# B&R Automation Studio project Assembly_and_ST (part 2)

#### providePellet.st
```iecst
ACTION providePellet:
		(*************************************************************************************************)
		(*************************************************************************************************)
		(* State Machine *)
	CASE gAssemblyModule.skill.providePellet.state.stateMachine.operationalState OF
		(*************************************************************************************************)
		(* RESETTING *)
		RESETTING:
			(*gAssemblyModule.skill.providePellet.state.stateMachine.stateTransition.reset := FALSE;*)

			IF gAssemblyModule.skill.providePellet.state.stateMachine.stateTransition.abort THEN
				gAssemblyModule.skill.providePellet.state.stateMachine.operationalState := ABORTING;

			ELSIF gAssemblyModule.skill.providePellet.state.stateMachine.stateTransition.stop THEN
				gAssemblyModule.skill.providePellet.state.stateMachine.operationalState := STOPPING;

			ELSE
				providePellet_Resetting;

			END_IF;

			(*************************************************************************************************)
			(* IDLE *)
		IDLE:

			gAssemblyModule.skill.providePellet.state.stateMachine.stateTransition.reset := FALSE;

			IF gAssemblyModule.skill.providePellet.state.stateMachine.stateTransition.abort THEN
				gAssemblyModule.skill.providePellet.state.stateMachine.operationalState := ABORTING;

			ELSIF gAssemblyModule.skill.providePellet.state.stateMachine.stateTransition.stop THEN
				gAssemblyModule.skill.providePellet.state.stateMachine.operationalState := STOPPING;

			ELSE
				providePellet_Idle;

			END_IF;

			(*************************************************************************************************)
			(* STARTING *)
		STARTING:
			(*gAssemblyModule.skill.providePellet.state.stateMachine.stateTransition.start := FALSE;*)

			IF gAssemblyModule.skill.providePellet.state.stateMachine.stateTransition.abort THEN
				gAssemblyModule.skill.providePellet.state.stateMachine.operationalState := ABORTING;

			ELSIF gAssemblyModule.skill.providePellet.state.stateMachine.stateTransition.stop THEN
				gAssemblyModule.skill.providePellet.state.stateMachine.operationalState := STOPPING;

			ELSE
				providePellet_Starting;

			END_IF;

			(*************************************************************************************************)
			(* RUNNING *)
		RUNNING:

			gAssemblyModule.skill.providePellet.state.stateMachine.stateTransition.start := FALSE;

			IF gAssemblyModule.skill.providePellet.state.stateMachine.stateTransition.abort THEN
				gAssemblyModule.skill.providePellet.state.stateMachine.operationalState := ABORTING;

			ELSIF gAssemblyModule.skill.providePellet.state.stateMachine.stateTransition.stop THEN
				gAssemblyModule.skill.providePellet.state.stateMachine.operationalState := STOPPING;

			ELSIF gAssemblyModule.skill.providePellet.state.stateMachine.stateTransition.hold THEN
				gAssemblyModule.skill.providePellet.state.stateMachine.operationalState := HOLDING;

			ELSIF gAssemblyModule.skill.providePellet.state.stateMachine.stateTransition.suspend THEN
				gAssemblyModule.skill.providePellet.state.stateMachine.operationalState := SUSPENDING;

			ELSIF gAssemblyModule.skill.providePellet.state.stateMachine.stateTransition.pause THEN
				gAssemblyModule.skill.providePellet.state.stateMachine.operationalState := PAUSING;

			ELSE
				providePellet_Running;

			END_IF;

			(*************************************************************************************************)
			(* PAUSING *)
		PAUSING:
			(*	gAssemblyModule.skill.providePellet.state.stateMachine.stateTransition.pause := FALSE;*)

			IF gAssemblyModule.skill.providePellet.state.stateMachine.stateTransition.abort THEN
				gAssemblyModule.skill.providePellet.state.stateMachine.operationalState := ABORTING;

			ELSIF gAssemblyModule.skill.providePellet.state.stateMachine.stateTransition.stop THEN
				gAssemblyModule.skill.providePellet.state.stateMachine.operationalState := STOPPING;

			ELSIF gAssemblyModule.skill.providePellet.state.stateMachine.stateTransition.hold THEN
				//gAssemblyModule.skill.providePellet.state.stateMachine.operationalState := HOLDING;

			ELSIF gAssemblyModule.skill.providePellet.state.stateMachine.stateTransition.suspend THEN
				//gAssemblyModule.skill.providePellet.state.stateMachine.operationalState := SUSPENDING;

			ELSE
				providePellet_Pausing;
			END_IF;

			(*************************************************************************************************)
			(* PAUSED *)
		PAUSED:

			gAssemblyModule.skill.providePellet.state.stateMachine.stateTransition.pause := FALSE;

			IF gAssemblyModule.skill.providePellet.state.stateMachine.stateTransition.abort THEN
				gAssemblyModule.skill.providePellet.state.stateMachine.operationalState := ABORTING;

			ELSIF gAssemblyModule.skill.providePellet.state.stateMachine.stateTransition.stop THEN
				gAssemblyModule.skill.providePellet.state.stateMachine.operationalState := STOPPING;

			ELSIF gAssemblyModule.skill.providePellet.state.stateMachine.stateTransition.hold THEN
				//gAssemblyModule.skill.providePellet.state.stateMachine.operationalState := HOLDING;

			ELSIF gAssemblyModule.skill.providePellet.state.stateMachine.stateTransition.suspend THEN
				//gAssemblyModule.skill.providePellet.state.stateMachine.operationalState := SUSPENDING;

			ELSE
				providePellet_Paused;

			END_IF;

			(*************************************************************************************************)
			(* SUSPENDING *)
		SUSPENDING:
			(*gAssemblyModule.skill.providePellet.state.stateMachine.stateTransition.suspend := FALSE;*)

			IF gAssemblyModule.skill.providePellet.state.stateMachine.stateTransition.abort THEN
				gAssemblyModule.skill.providePellet.state.stateMachine.operationalState := ABORTING;

			ELSIF gAssemblyModule.skill.providePellet.state.stateMachine.stateTransition.stop THEN
				gAssemblyModule.skill.providePellet.state.stateMachine.operationalState := STOPPING;

			ELSIF gAssemblyModule.skill.providePellet.state.stateMachine.stateTransition.hold THEN
				//gAssemblyModule.skill.providePellet.state.stateMachine.operationalState := HOLDING;

			ELSE
				providePellet_Suspending;

			END_IF;

			(*************************************************************************************************)
			(* SUSPENDED *)
		SUSPENDED:

			gAssemblyModule.skill.providePellet.state.stateMachine.stateTransition.suspend := FALSE;

			IF gAssemblyModule.skill.providePellet.state.stateMachine.stateTransition.abort THEN
				gAssemblyModule.skill.providePellet.state.stateMachine.operationalState := ABORTING;

			ELSIF gAssemblyModule.skill.providePellet.state.stateMachine.stateTransition.stop THEN
				gAssemblyModule.skill.providePellet.state.stateMachine.operationalState := STOPPING;

			ELSIF gAssemblyModule.skill.providePellet.state.stateMachine.stateTransition.hold THEN
				//gAssemblyModule.skill.providePellet.state.stateMachine.operationalState := HOLDING;

			ELSE
				providePellet_Suspended;

			END_IF;

			(*************************************************************************************************)
			(* UNSUSPENDING *)
		UNSUSPENDING:
			gAssemblyModule.skill.providePellet.state.stateMachine.stateTransition.unsuspend := FALSE;

			IF gAssemblyModule.skill.providePellet.state.stateMachine.stateTransition.abort THEN
				gAssemblyModule.skill.providePellet.state.stateMachine.operationalState := ABORTING;

			ELSIF gAssemblyModule.skill.providePellet.state.stateMachine.stateTransition.stop THEN
				gAssemblyModule.skill.providePellet.state.stateMachine.operationalState := STOPPING;

			ELSIF gAssemblyModule.skill.providePellet.state.stateMachine.stateTransition.hold THEN
				//gAssemblyModule.skill.providePellet.state.stateMachine.operationalState := HOLDING;

			ELSE
				providePellet_Unsuspending;

			END_IF;

			(*************************************************************************************************)
			(* HOLDING *)
		HOLDING:
			(*gAssemblyModule.skill.providePellet.state.stateMachine.stateTransition.hold := FALSE;*)

			IF gAssemblyModule.state.stateMachine.stateTransition.abort THEN
				gAssemblyModule.state.stateMachine.operationalState := ABORTING;

			ELSIF gAssemblyModule.state.stateMachine.stateTransition.stop THEN
				gAssemblyModule.state.stateMachine.operationalState := STOPPING;

			ELSE
				providePellet_Holding;

			END_IF;

			(*************************************************************************************************)
			(* HELD *)
		HELD:

			gAssemblyModule.skill.providePellet.state.stateMachine.stateTransition.hold := FALSE;

			IF gAssemblyModule.skill.providePellet.state.stateMachine.stateTransition.abort THEN
				gAssemblyModule.skill.providePellet.state.stateMachine.operationalState := ABORTING;

			ELSIF gAssemblyModule.skill.providePellet.state.stateMachine.stateTransition.stop THEN
				gAssemblyModule.skill.providePellet.state.stateMachine.operationalState := STOPPING;

			ELSE
				providePellet_Held;

			END_IF;

			(*************************************************************************************************)
			(* UNHOLDING *)
		UNHOLDING:
			gAssemblyModule.skill.providePellet.state.stateMachine.stateTransition.unhold := FALSE;

			IF gAssemblyModule.skill.providePellet.state.stateMachine.stateTransition.abort THEN
				gAssemblyModule.skill.providePellet.state.stateMachine.operationalState := ABORTING;

			ELSIF gAssemblyModule.skill.providePellet.state.stateMachine.stateTransition.stop THEN
				gAssemblyModule.skill.providePellet.state.stateMachine.operationalState := STOPPING;

			ELSE
				providePellet_Unholding;

			END_IF;

			(*************************************************************************************************)
			(* COMPLETING *)
		COMPLETING:

			IF gAssemblyModule.skill.providePellet.state.stateMachine.stateTransition.abort THEN
				gAssemblyModule.skill.providePellet.state.stateMachine.operationalState := ABORTING;

			ELSIF gAssemblyModule.skill.providePellet.state.stateMachine.stateTransition.stop THEN
				gAssemblyModule.skill.providePellet.state.stateMachine.operationalState := STOPPING;

			ELSE
				providePellet_Completing;

			END_IF;

			(*************************************************************************************************)
			(* COMPLETE *)
		COMPLETE:

			IF gAssemblyModule.skill.providePellet.state.stateMachine.stateTransition.abort THEN
				gAssemblyModule.skill.providePellet.state.stateMachine.operationalState := ABORTING;

			ELSIF gAssemblyModule.skill.providePellet.state.stateMachine.stateTransition.stop THEN
				gAssemblyModule.skill.providePellet.state.stateMachine.operationalState := STOPPING;

			ELSE
				providePellet_Complete;

			END_IF;

			(*************************************************************************************************)
			(* STOPPING *)
		STOPPING:
			(*gAssemblyModule.skill.providePellet.state.stateMachine.stateTransition.stop := FALSE;*)

			IF gAssemblyModule.skill.providePellet.state.stateMachine.stateTransition.abort THEN
				gAssemblyModule.skill.providePellet.state.stateMachine.operationalState := ABORTING;

			ELSE
				providePellet_Stopping;

			END_IF;

			(*************************************************************************************************)
			(* STOPPED *)
		STOPPED:

			gAssemblyModule.skill.providePellet.state.stateMachine.stateTransition.stop := FALSE;

			IF gAssemblyModule.skill.providePellet.state.stateMachine.stateTransition.abort THEN
				gAssemblyModule.skill.providePellet.state.stateMachine.operationalState := ABORTING;

			ELSE
				providePellet_Stopped;

			END_IF;

			(*************************************************************************************************)
			(* ABORTING *)
		ABORTING:
			(*gAssemblyModule.skill.providePellet.state.stateMachine.stateTransition.abort := FALSE;*)

			providePellet_Aborting;

			(*************************************************************************************************)
			(* ABORTED *)
		ABORTED:

			gAssemblyModule.skill.providePellet.state.stateMachine.stateTransition.abort := FALSE;

			providePellet_Aborted;

			(*************************************************************************************************)
			(* CLEARING *)
		CLEARING:
			gAssemblyModule.skill.providePellet.state.stateMachine.stateTransition.clear := FALSE;

			providePellet_Clearing;

			(*************************************************************************************************)
			(* ELSE *)
		ELSE;

	END_CASE;
END_ACTION
```

#### providePellet_Clearing.st
```iecst
ACTION providePellet_Clearing:

	gAssemblyModule.skill.providePellet.state.stateMachine.stateTransition.clear := FALSE;

	gAssemblyModule.skill.providePellet.state.stateMachine.operationalState := STOPPED;

END_ACTION
```

#### providePellet_Idle.st
```iecst
ACTION providePellet_Idle:

	IF gAssemblyModule.skill.providePellet.state.stateMachine.stateTransition.start THEN
			gAssemblyModule.skill.providePellet.state.stateMachine.operationalState := STARTING;

	END_IF

END_ACTION
```

#### providePellet_Starting.st
```iecst
ACTION providePellet_Starting:

	gAssemblyModule.skill.providePellet.state.stateMachine.operationalState := RUNNING;

END_ACTION
```

#### providePellet_Completing.st
```iecst
ACTION providePellet_Completing:

	providePellet_Case := PELLET_SUPPLY_DECISION_CASE;
	gAssemblyModule.skill.providePellet.inputParameters.pelletType :=0;
	gAssemblyModule.skill.providePellet.state.stateMachine.operationalState := COMPLETE;

END_ACTION
```

#### providePellet_Complete.st
```iecst
ACTION providePellet_Complete:

	Checked := FALSE;
	IF gAssemblyModule.skill.providePellet.state.stateMachine.stateTransition.reset THEN
		gAssemblyModule.skill.providePellet.state.stateMachine.operationalState := RESETTING;
	END_IF;

END_ACTION
```

#### providePellet_Holding.st
```iecst
ACTION providePellet_Holding:

	gAssemblyModule.skill.providePellet.state.stateMachine.operationalState := HELD;

END_ACTION
```

#### providePellet_Unholding.st
```iecst
ACTION providePellet_Unholding:

		gAssemblyModule.skill.providePellet.state.stateMachine.operationalState := RUNNING;

END_ACTION
```

#### providePellet_Suspending.st
```iecst
ACTION providePellet_Suspending:

	gAssemblyModule.skill.providePellet.state.stateMachine.operationalState := SUSPENDED;

END_ACTION
```

#### providePellet_Suspended.st
```iecst
ACTION providePellet_Suspended:

	IF gAssemblyModule.skill.providePellet.state.stateMachine.stateTransition.unsuspend THEN
		gAssemblyModule.skill.providePellet.state.stateMachine.operationalState := UNSUSPENDING;
	END_IF;

END_ACTION
```

#### providePellet_Unsuspending.st
```iecst
ACTION providePellet_Unsuspending:

	gAssemblyModule.skill.providePellet.state.stateMachine.operationalState := RUNNING;

END_ACTION
```

### MNG_Global.typ - Global data types
```iecst
(*                                                                            *)
(* File generated by the B&R AS 4 control config generator                    *)
(*                                                                            *)
(*     Provider: machineering                                                 *)
(*  Application: industrialPhysics                                            *)
(* Architecture: Windows 64 Bit                                               *)
(*      Version: 2.2.8481.master                                              *)
(*        Build: 057354c2a                                                    *)
(*         Date: 2020-02-28, Time: 15:09:14                                   *)
(*                                                                            *)

TYPE
    (* 3d position *)
    VEC3 : STRUCT
                    x: REAL;
                    y: REAL;
                    z: REAL;
    END_STRUCT;

    (* position and orientation as an euler based pose *)
    POSE6 :	STRUCT
                    x: REAL;
                    y: REAL;
                    z: REAL;
                    a: REAL;
                    b: REAL;
                    c: REAL;
    END_STRUCT;

    (* position and orientation as a 4x4 matrix *)
    TRAFO :STRUCT
                    baseX : VEC3;
                    fill0 : REAL;
                    baseY : VEC3;
                    fill1 : REAL;
                    baseZ : VEC3;
                    fill2 : REAL;
                    origin : VEC3;
                    fill3 : REAL;
    END_STRUCT;

                MNG_APPLICATION_INPUTS_32BIT : STRUCT
    NumSignals                    : INT     := 3         ;
    Gripper01_VACUUM                : BOOL    := 0; (* omau_Link5_Comau_Link6_Gripper_Comau_Gripper?Vacuum *)
    PaperCupDrawer01_IsOpened       : BOOL    := 0; (* embly_Module_PaperCupSupply_PaperCupDrawer?IsOpened *)
    PlasticCupDrawer01_IsOpened     : BOOL    := 0; (* y_Module_PlasticCupSupply_PlasticCupDrawer?IsOpened *)
END_STRUCT;
MNG_APPLICATION_OUTPUTS_32BIT : STRUCT
    NumSignals                    : INT     := 9         ;
    Comau_Link101_TGT_POS           : REAL    := 0.0; (* _Assembly_Module_Comau_Racer3_Comau_Link1?KinTarget *)
    Comau_Link201_TGT_POS           : REAL    := 0.0; (* dule_Comau_Racer3_Comau_Link1_Comau_Link2?KinTarget *)
    Comau_Link301_TGT_POS           : REAL    := 0.0; (* acer3_Comau_Link1_Comau_Link2_Comau_Link3?KinTarget *)
    Comau_Link401_TGT_POS           : REAL    := 0.0; (* Link1_Comau_Link2_Comau_Link3_Comau_Link4?KinTarget *)
    Comau_Link501_TGT_POS           : REAL    := 0.0; (* Link2_Comau_Link3_Comau_Link4_Comau_Link5?KinTarget *)
    Comau_Link601_TGT_POS           : REAL    := 0.0; (* Link3_Comau_Link4_Comau_Link5_Comau_Link6?KinTarget *)
    Gripper01_GRIP                  : BOOL    := 0; (* mau_Link5_Comau_Link6_Gripper_Comau_Gripper?Gripper *)
    PaperCupDrawer01_Assem          : BOOL    := 0; (* ssembly_Module_PaperCupSupply_PaperCupDrawer?_Assem *)
    PlasticCupDrawer01_Assem        : BOOL    := 0; (* bly_Module_PlasticCupSupply_PlasticCupDrawer?_Assem *)
END_STRUCT;

END_TYPE
```

### Program Logical/Assembly_Module/MNG_Interface (IEC) - Programm

#### MNG_Interface.fun
```iecst
(********************************************************************
 * COPYRIGHT 2014 machineering GmbH & Co. KG
 ********************************************************************
 * Programm: MNG_Interface
 * Datei: MNG_Interface.fun
 * Autor: machineering GmbH & Co. KG
 * Erstellt: 24. Februar 2014
 ********************************************************************
 * Funktionen und Funktionsblöcke des Programmes MNG_Interface
 ********************************************************************)

FUNCTION_BLOCK MNG_COPY_MSG_TO_INPUTS
	VAR_OUTPUT
		Counter : UDINT;
		Success : BOOL;
	END_VAR
	VAR_IN_OUT
		fromServer : MNG_RawDatagram;
		inputs : MNG_APPLICATION_INPUTS_32BIT;
	END_VAR
	VAR
		datagramType : MNG_DatagramType;
		DWordBuffer : UDINT; (* convert DWORD data *)
		DIntBuffer : DINT; (* convert DINT data *)
		byteCount : UDINT;
		numSignalsInMessage : UDINT;
	END_VAR
END_FUNCTION_BLOCK

FUNCTION_BLOCK MNG_COPY_OUTPUTS_INTO_MSG (*TODO: Bitte Kommentar hier einfügen*) (*$GROUP=Anwender*)
	VAR_INPUT
		Counter : UDINT;
	END_VAR
	VAR_IN_OUT
		toServer : MNG_RawDatagram;
		outputs : MNG_APPLICATION_OUTPUTS_32BIT;
	END_VAR
	VAR
		DWordBuffer : UDINT; (* convert DWORD data *)
		DIntBuffer : DINT; (* convert DINT data *)
	END_VAR
END_FUNCTION_BLOCK
```

#### MNG_COPY_MSG_TO_INPUTS.st
```iecst
(*                                                                            *)
(* File generated by the B&R AS 4 control config generator                    *)
(*                                                                            *)
(*     Provider: machineering                                                 *)
(*  Application: industrialPhysics                                            *)
(* Architecture: Windows 64 Bit                                               *)
(*      Version: 2.2.8481.master                                              *)
(*        Build: 057354c2a                                                    *)
(*         Date: 2020-02-28, Time: 15:09:14                                   *)
(*                                                                            *)
FUNCTION_BLOCK MNG_COPY_MSG_TO_INPUTS

    byteCount := N_TO_HUDINT(fromServer.Header.ByteCount);
    datagramType := N_TO_HUDINT(fromServer.Header.DatagramType);
    IF datagramType <> MNG_Raw32BitImage THEN
        Success := FALSE;
        RETURN;
    END_IF

    inputs.NumSignals := 3;

    numSignalsInMessage := N_TO_HUDINT(fromServer.Payload[1]);
    IF UDINT_TO_DINT(numSignalsInMessage) <> inputs.NumSignals OR byteCount <> 4 + numSignalsInMessage * 4	THEN
            Success := FALSE;
            RETURN;
    END_IF

    Counter := N_TO_HUDINT(fromServer.Header.Counter);

    (* BOOL Gripper01_VACUUM *)
    inputs.Gripper01_VACUUM := fromServer.Payload[2]<>0;

    (* BOOL PaperCupDrawer01_IsOpened *)
    inputs.PaperCupDrawer01_IsOpened := fromServer.Payload[3]<>0;

    (* BOOL PlasticCupDrawer01_IsOpened *)
    inputs.PlasticCupDrawer01_IsOpened := fromServer.Payload[4]<>0;

END_FUNCTION_BLOCK
```

### SuperTrak_Global.var
```iecst
(*======================================*)
(*SuperTrak module type*)
(*======================================*)
VAR
	gSuperTrak : opcSuperTrakType;
END_VAR
(*======================================*)
(*Function blocks*)
(*======================================*)
VAR
	StSection_ : ARRAY[1..SUPERTRAK_SECTIONS] OF StSection;
	StSectionCtrl_ : ARRAY[1..SUPERTRAK_SECTIONS] OF StSection;
	StControl_0 : StControl;
	StTargetExt_ : ARRAY[1..SUPERTRAK_TARGETS] OF StTargetExt;
END_VAR
(*======================================*)
(*Control parameters*)
(*======================================*)
VAR
	SuperTrakSectionParameters : StSectionParType;
	SuperTrakControlParameters : StControlParType;
	TargetControlParameters : ARRAY[1..SUPERTRAK_TARGETS] OF StTargetExtParType;
END_VAR
(*======================================*)
(*Variables for Event ID's in alarm management*)
(*======================================*)
VAR
	QA_Door_Closed : BOOL;
	Severity_Code : USINT; (*Severity of the message ( success, info, warning or error)*)
	Facility_Code : UINT; (*Facility in which the error was produced*)
	Code : UINT; (*Error code with value between 0 and 65535*)
END_VAR
(*
 ********************************************************************
 * Global Supertrak Variables
 ********************************************************************)
(*Global variable for internal use*)
VAR
	gStLink : {REDUND_UNREPLICABLE} StLinkType := (0); (*StCom library communication variable*)
END_VAR
(************************************************************************************************************************************)
(************************************************************************************************************************************)
(*Global variables for communication to/from SuperTrak*)
VAR
	gStCyclicControlData : {REDUND_UNREPLICABLE} ARRAY[0..499] OF USINT := [500(0)]; (*Cyclic control buffer (to SuperTrak)*)
	gStCyclicStatusData : {REDUND_UNREPLICABLE} ARRAY[0..499] OF USINT := [500(0)]; (*Cyclic status buffer (from SuperTrak)*)
	gStServiceChannelReqData : {REDUND_UNREPLICABLE} ARRAY[0..127] OF USINT := [128(0)]; (*Service channel request buffer (to SuperTrak)*)
	gStServiceChannelResData : {REDUND_UNREPLICABLE} ARRAY[0..127] OF USINT := [128(0)]; (*Service channel response buffer (from SuperTrak)*)
END_VAR
(************************************************************************************************************************************)
(************************************************************************************************************************************)
VAR
	ST_LightBarrier_E2_E : BOOL;
	ST_LightBarrier_E1_E : BOOL;
	ST_LightBarrier_ContactComprob_R : BOOL;
	ST_LightBarrier_ConfirmInput_R : BOOL;
	ST_LightBarrier_Signal_R : BOOL;
	ST_LightBarrier_SecurityOut1_R : BOOL;
	ST_LightBarrier_SecurityOut2_R : BOOL;
	Disable_Light_Barrier : BOOL;
END_VAR
(*Insert your comment here.*)
(*Insert your comment here.*)
VAR
	LED_Green : BOOL;
	LED_Blue : BOOL;
	LED_Red : BOOL;
	Outfeed_LED_Green : BOOL;
	Outfeed_LED_Blue : BOOL;
	Outfeed_LED_Red : BOOL;
	Outfeed_Full : BOOL;
	QA_Actuator_UP : BOOL;
	QA_Actuator_DOWN : BOOL;
	Outfeed_Actuator_FRONT : BOOL;
	Outfeed_Actuator_BACK : BOOL;
	Outfeed_Actuator_UP : BOOL;
	Outfeed_Actuator_DOWN : BOOL;
END_VAR
```

### Program Logical/SuperTrak_Module/ST_Main

#### Main.st
```iecst
(*********************************************************************************
 * Copyright: ATS Automation Tooling Systems, Inc. 2015
 *     All rights reserved.
 *********************************************************************************
 *********************************************************************************
 * Description:
 * -------------------------------------------------------------------------------
 * This task configures the internal communication structure AND controlls
 * the SuperTrak system.
 *********************************************************************************)

PROGRAM _INIT

 // SuperTrak initialization
	IF DiagCpuIsSimulated() THEN
		SuperTrakInit(TRUE,'/DEVICE=C:\GIT\Assembly_and_Supertrak\plc-code\SuperTrakUser');
//		SuperTrakInit(TRUE,'/DEVICE=C:\Users\guelmez\Documents\Implementation\SuperTrakUser');
	ELSE
		//This is the user partition of the cf card used into the IPC
		SuperTrakInit(FALSE,'/DEVICE=F:');
	END_IF;

	// Service Channel initialization
	ServiceChannelData.channelId      := 1;
	ServiceChannelData.pRequestHeader  := ADR(gStServiceChannelReqData);
	ServiceChannelData.pResponseHeader  := ADR(gStServiceChannelResData);
	ServiceChannelData.pRequestValues      := ADR(gStServiceChannelReqData) + SIZEOF(ServiceChannelHeader_t);
	ServiceChannelData.pResponseValues     := ADR(gStServiceChannelResData) + SIZEOF(ServiceChannelHeader_t);
	ServiceChannelData.requestBufferSize   := SIZEOF(gStServiceChannelReqData);
	ServiceChannelData.responseBufferSize   := SIZEOF(gStServiceChannelResData);
	ServiceChannelData.state        := scSTATE_RECV;

	pResView ACCESS ADR(gStServiceChannelResData);
	pReqView ACCESS ADR(gStServiceChannelReqData);

	// Command interface mapping
	SuperTrakControlInterface[0].pControl   := ADR(gStCyclicControlData);
	SuperTrakControlInterface[0].pStatus    := ADR(gStCyclicStatusData);
	SuperTrakControlInterface[0].controlSize:= SIZEOF(gStCyclicControlData);
	SuperTrakControlInterface[0].statusSize := SIZEOF(gStCyclicStatusData);

END_PROGRAM

PROGRAM _CYCLIC

 // Cylcic SuperTrak control
	SuperTrakCyclic();

	// Map internal communication structure
	FOR i := 0 TO stMAX_CONTROL_IF_INDEX DO
		SuperTrakProcessControl(i, SuperTrakControlInterface[i]);
	END_FOR;

	// Service channel handling
	IF ServiceChannelData.state = scSTATE_RECV AND
		pReqView.sequence <> pResView.sequence THEN
		ServiceChannelData.requestSequence  := pReqView.sequence;
		ServiceChannelData.state    := scSTATE_EXEC;
	ELSIF ServiceChannelData.state = scSTATE_EXEC OR ServiceChannelData.state = scSTATE_WAIT THEN
		SuperTrakServiceChannel(ServiceChannelData);
	ELSIF ServiceChannelData.state = scSTATE_SEND THEN
		ServiceChannelData.state    := scSTATE_RECV;
	END_IF;

END_PROGRAM

PROGRAM _EXIT

 // Clear internal memory
	SuperTrakExit();

END_PROGRAM
```

### Program Logical/SuperTrak_Module/ST_Visu

#### Types.typ
```iecst
TYPE
	RoboVisuPallet_t : 	STRUCT
		Visible : BOOL; (*byte 0*)
		reserved_1 : USINT; (*byte 1*)
		Text : STRING[5]; (*Text / bytes 2-7*) (*STRING[n] = char[n + 1] = n characters plus terminator*)
		X : REAL; (*Position.X / bytes 8-11*)
		Y : REAL; (*Position.Y / bytes 12-15*)
		RZ : REAL; (*Orientation.RotZ / bytes 16-19*)
	END_STRUCT;
	RoboVisuData_t : 	STRUCT
		StraightSectionVisible : ARRAY[0..63]OF BOOL; (*bytes 0-63*)
		N180SectionVisible : ARRAY[0..1]OF BOOL; (*bytes 64-65*)
		W180SectionVisible : ARRAY[0..1]OF BOOL; (*bytes 66-67*)
		StraightSectionPositionY : REAL; (*bytes 68-71*)
		CurvePositionX : REAL; (*bytes 72-75*)
		reserved_76 : REAL; (*bytes 76-79*)
		reserved_80 : ARRAY[0..47]OF USINT; (*bytes 80-127*)
		reserved_128 : ARRAY[0..383]OF USINT; (*bytes 128-511*)
		Pallet : ARRAY[0..127]OF RoboVisuPallet_t; (*bytes 512-3071*)
	END_STRUCT;
	SectionInfo_t : 	STRUCT
		userAddress : UINT;
		sectionType : UINT;
		side : INT;
		modelIndex : INT;
		positionX : REAL;
	END_STRUCT;
END_TYPE
```

#### Main.st
```iecst
(*********************************************************************************
 * Copyright Bernecker + Rainer 2015
 * Copyright ATS Automation Tooling Systems, Inc. 2017-2018
 * All rights reserved.
 * -------------------------------------------------------------------------------
 * This task calculates the actual pallet positions in the room based on the
 * section number and the position of the pallet in the section.
 * It is also hiding unused sections and/or pallets.
 * This data is then provided to B&R Scene Viewer.
 *********************************************************************************)

PROGRAM _INIT

	visuStep := 0;

END_PROGRAM

PROGRAM _CYCLIC

	CASE visuStep OF
		visuSTEP_INITIALIZE:
			visuStep := visuSTEP_GET_SECTION_COUNT;

		visuSTEP_GET_SECTION_COUNT:
			// read parameter 1080: section count
			result := SuperTrakServChanRead(0, 1080, 0, 1, ADR(sectionCount), SIZEOF(sectionCount));

			IF (result = scERR_SUCCESS) AND (sectionCount > 0) THEN
				visuStep := visuSTEP_GET_SECTION_ADDRS;
			ELSE
				visuStep := visuSTEP_ERROR;
			END_IF;

		visuSTEP_GET_SECTION_ADDRS:
			// read parameter 1081: section user address
			result := SuperTrakServChanRead(0, 1081, 0, sectionCount, ADR(servChanResponseUINT), SIZEOF(servChanResponseUINT));

			IF (result = scERR_SUCCESS) THEN
				FOR i := 0 TO sectionCount - 1 DO
					Section[i].userAddress := servChanResponseUINT[i];

					IF (Section[i].userAddress > 0) AND (Section[i].userAddress < 99) THEN
						sectionLookup[ Section[i].userAddress ] := i;
					END_IF;
				END_FOR;

				visuStep := visuSTEP_GET_SECTION_TYPES;
				i := 0;
			ELSE
				visuStep := visuSTEP_ERROR;
			END_IF;

		visuSTEP_GET_SECTION_TYPES:
			// read parameter 1082: section type
			result := SuperTrakServChanRead(UINT_TO_USINT(Section[i].userAddress), 1082, 0, 1, ADR(Section[i].sectionType), SIZEOF(UINT));

			IF (result = scERR_SUCCESS) THEN
				i := i + 1;

				IF (i >= sectionCount) THEN
					visuStep := visuSTEP_SETUP_SECTIONS;
				END_IF;
			ELSE
				visuStep := visuSTEP_ERROR;
			END_IF;

		visuSTEP_SETUP_SECTIONS:
			// Assign visualization models to sections.
			// Mostly assume that the layout is sensible.
			side := 0;
			sideLength[0] := 0;
			sideLength[1] := 0;
			position := 0;
			modelIndex := 0;

			FOR i := 0 TO sectionCount - 1 DO
				Section[i].side := -1;
				Section[i].modelIndex := -1;

				IF (Section[i].sectionType = SECTION_TYPE_1M) OR (Section[i].sectionType = SECTION_TYPE_1M_LP) THEN
					// Straight section models are indexed 0-31 (front) and 32-63 (back).
					IF (side < 2)
						AND (modelIndex >= (side * 32))
						AND (modelIndex < ((side + 1) * 32)) THEN

						Section[i].side := side;
						sideLength[side] := sideLength[side] + 1;

						Data.StraightSectionVisible[modelIndex] := TRUE;
						Section[i].modelIndex := modelIndex;
						modelIndex := modelIndex + 1;

						Section[i].positionX := position;

						IF (side = 0) THEN
							position := position + 1000;
						ELSE
							position := position - 1000;
						END_IF;
					END_IF;

				ELSIF (Section[i].sectionType = SECTION_TYPE_N180) OR (Section[i].sectionType = SECTION_TYPE_W180L) THEN
					// Advance to next side when a curve follows straights,
					// or when a curve already exists on the current side.
					IF (side < 2) AND ((sideLength[side] > 0) OR (curveHSection[side] >= 0)) THEN
						side := side + 1;

						IF (side = 1) THEN
							modelIndex := 64 - sideLength[0];
							Data.CurvePositionX := position;
						END_IF;
					END_IF;

					IF (side = 1) THEN
						curveSide := 1;
					ELSE
						curveSide := 0;
					END_IF;

					IF (curveHSection[curveSide] < 0) THEN
						Section[i].side := curveSide;
						curveHSection[curveSide] := i;

						IF (Section[i].sectionType = SECTION_TYPE_N180) THEN
							Data.N180SectionVisible[curveSide] := TRUE;
						ELSE
							Data.W180SectionVisible[curveSide] := TRUE;
						END_IF;

						curveType := Section[i].sectionType;
					END_IF;

				ELSIF (Section[i].sectionType = SECTION_TYPE_W180R) THEN
					IF (side = 1) THEN
						curveSide := 1;
					ELSE
						curveSide := 0;
					END_IF;

					Section[i].side := curveSide;

				ELSE
					// unhandled section type

				END_IF;
			END_FOR;

			IF (curveType = SECTION_TYPE_N180) THEN
				Data.StraightSectionPositionY := 0;
				straightPalletPositionY[0] := -236;
				straightPalletPositionY[1] := 236;
			ELSE // W180
				Data.StraightSectionPositionY := 365.5;
				straightPalletPositionY[0] := -236;
				straightPalletPositionY[1] := 600.5;
			END_IF;

			visuStep := visuSTEP_RUN;

		visuSTEP_RUN:
			// get actual pallet positions
			SuperTrakGetPalletInfo(ADR(Pallet), 128, FALSE);

			FOR i := 0 TO 127 DO
				IF (Pallet[i].section >= 1) AND (Pallet[i].section <= 99) THEN
					h := sectionLookup[ Pallet[i].section ];
				ELSE
					h := -1;
				END_IF;

				IF (h >= 0) THEN
					// display this pallet
					Data.Pallet[i].Visible := TRUE;
					position := DINT_TO_REAL(Pallet[i].position) / 1000;

					IF (Section[h].sectionType = SECTION_TYPE_1M) OR (Section[h].sectionType = SECTION_TYPE_1M_LP) THEN
						IF (Section[h].side = 0) THEN
							Data.Pallet[i].X := Section[h].positionX + position;
							Data.Pallet[i].Y := straightPalletPositionY[0];
							Data.Pallet[i].RZ := 0;
						ELSE
							Data.Pallet[i].X := Section[h].positionX - position;
							Data.Pallet[i].Y := straightPalletPositionY[1];
							Data.Pallet[i].RZ := 180;
						END_IF;

					ELSIF (Section[h].sectionType = SECTION_TYPE_N180) THEN
						// approximate the shape of the curve
						IF (position <= 15) THEN
							Data.Pallet[i].X := position;
							Data.Pallet[i].Y := -236;
							Data.Pallet[i].RZ := 0;
						ELSIF (position < 1015) THEN
							angle := brmPI * (position - 15) / 1000;
							Data.Pallet[i].X := 15 + (355 * SIN(angle)) - (15 * SIN(angle * 3));
							Data.Pallet[i].Y := (-257 * COS(angle)) + (21 * COS(angle * 3));
							Data.Pallet[i].RZ := 90 - 90 * COS(angle);
						ELSE
							Data.Pallet[i].X := 1030 - position;
							Data.Pallet[i].Y := 236;
							Data.Pallet[i].RZ := 180;
						END_IF;

						IF (Section[h].side = 0) THEN
							Data.Pallet[i].X := -Data.Pallet[i].X;
							Data.Pallet[i].Y := -Data.Pallet[i].Y;
							Data.Pallet[i].RZ := Data.Pallet[i].RZ - 180;
						ELSE
							Data.Pallet[i].X := Data.Pallet[i].X + Data.CurvePositionX;
						END_IF;

					ELSIF (Section[h].sectionType = SECTION_TYPE_W180L) THEN
						IF (position > 100) THEN
							angle := (position - 100) / W180_RADIUS * 180 / brmPI;
							position := 100;
						ELSE
							angle := 0;
						END_IF;

						IF (Section[h].side = 0) THEN
							Data.Pallet[i].X := -position - W180_RADIUS * SIN(angle * brmPI / 180);
							Data.Pallet[i].Y := 181.75 + W180_RADIUS * COS(angle * brmPI / 180);
							angle := angle + 180;
						ELSE
							Data.Pallet[i].X := position + Data.CurvePositionX + W180_RADIUS * SIN(angle * brmPI / 180);
							Data.Pallet[i].Y := 181.75 - W180_RADIUS * COS(angle * brmPI / 180);
						END_IF;

						Data.Pallet[i].RZ := angle;

					ELSIF (Section[h].sectionType = SECTION_TYPE_W180R) THEN
						IF (position > 650) THEN
							angle := 180;
							position := 750 - position;
						ELSE
							angle := (position / W180_RADIUS * 180 / brmPI) + 90;
							position := 100;
						END_IF;

						IF (Section[h].side = 0) THEN
							angle := angle + 180;
							Data.Pallet[i].X := -position - W180_RADIUS * ABS(SIN(angle * brmPI / 180));
							Data.Pallet[i].Y := 181.75 - W180_RADIUS * ABS(COS(angle * brmPI / 180));
						ELSE
							Data.Pallet[i].X := position + Data.CurvePositionX + W180_RADIUS * ABS(SIN(angle * brmPI / 180));
							Data.Pallet[i].Y := 181.75 + W180_RADIUS * ABS(COS(angle * brmPI / 180));
						END_IF;

						Data.Pallet[i].RZ := angle;

					END_IF;

				ELSE
					// hide this pallet
					Data.Pallet[i].Visible := FALSE;
					Data.Pallet[i].X := 0;
					Data.Pallet[i].Y := 0;
					Data.Pallet[i].RZ := 0;

				END_IF;
			END_FOR;

		ELSE
			// error or unhandled state; do nothing

	END_CASE;

END_PROGRAM
```

### Program Logical/SuperTrak_Module/StateMachine_SuperTrak (IEC)

#### Types.typ - Local data types
```iecst
TYPE
	Calibration_Enum :
		(
		ENABLE_SYSTEM,
		ID_SETTING,
		SEND_TO_QA,
		ABORTED_RESET_POSITIONS,
		ABORTED_CALIBRATION,
		ABORTED_SEND_TO_QA,
		CALIBRATION_END
		);
END_TYPE
```

#### Variables.var - Local variables
```iecst
(*==============================================*)
(*Process control variables*)
(*==============================================*)
VAR
	Calibration_Finished : BOOL;
	Shuttle_sent : USINT;
	MES_Test : BOOL;
	first_shuttle : BOOL;
	Skills_Aborted : USINT;
	Aborting_Init : BOOL;
	Transition_From_Stopped : BOOL;
	transitionFromAborted : BOOL;
	QA_finished : BOOL;
END_VAR
(*==============================================*)
(*Indexes for internal code use*)
(*==============================================*)
VAR
	New_ID : USINT;
	First_ID : USINT;
	Last_ID : USINT;
	Shuttle : USINT := 0;
	shuttleCounter : USINT;
	Last_Shuttle : DINT;
	Index : USINT;
	iShuttle : USINT;
	iMessageHelper : USINT := 0; (* Calibration *)
	Identifier : STRING[80];
	j : USINT;
	i : ARRAY[1..6] OF USINT;
	Checking : BOOL;
END_VAR
(*==============================================*)
(*Calibration state machine*)
(*==============================================*)
VAR
	Calibration_State : Calibration_Enum;
END_VAR
(*==============================================*)
(*Process Timers*)
(*==============================================*)
VAR
	Counter_Check_Shuttle : TON;
	Counter_Clearing_Timeout : TON;
	Time_For_AbortClearing_Start : TON;
	Time_For_AbortClearing_End : TON;
	Time_For_Stop : TON;
	Timer_Send_Super_Trak_In_Stop : TON;
	check_Parking_Timeout : TON;
	Timer_Outfeed_FRONT : TON;
	Timer_Outfeed_BACK : TON;
	Timer_Outfeed_DOWN : TON;
	Timer_Outfeed_UP : TON;
	Timer_Actuator_UP : TON;
	Timer_Enable_Barrier : TON;
	Timer_Actuator_DOWN : TON;
END_VAR
(*==============================================*)
(*Aborted Calibration options*)
(*==============================================*)
VAR
	SetID : BOOL;
END_VAR
```

#### Aborting.st
```iecst
ACTION Aborting:

	Counter_Clearing_Timeout(IN:= FALSE);
	Last_Shuttle := -1;

	//Disable all sections
	StControl_0.EnableAllSections := FALSE;

	Calibration_State := ENABLE_SYSTEM;

	//Send abort transition to the skills
	gSuperTrak.skill.checkParking.state.stateMachine.stateTransition.abort := TRUE;
	gSuperTrak.skill.QACheck.state.stateMachine.stateTransition.abort := TRUE;
	gSuperTrak.skill.Outfeed.state.stateMachine.stateTransition.abort := TRUE;

	FOR iShuttle := 1 TO SUPERTRAK_SHUTTLES DO
		gSuperTrak.skill.moveShuttle[iShuttle].state.stateMachine.stateTransition.abort := TRUE;
	END_FOR;

	//Wait for the sections to be disabled and skills to be aborted and then go into aborted state
	IF NOT StControl_0.SectionsEnabled AND Skills_Aborted = (SUPERTRAK_SKILLS) THEN

		gSuperTrak.state.stateMachine.operationalState := ABORTED;

	END_IF;

END_ACTION
```

#### Aborted.st
```iecst
ACTION Aborted:

	(* Reset MessageSum *)
	transitionFromAborted := TRUE;
	(* Checking all errors for TRUE State --> If: SumCritical is TRUE, if not: SumCritical is FALSE *)
	Timer_Actuator_DOWN (IN:= FALSE);
	Timer_Actuator_UP (IN:= FALSE);

	Skills_Aborted := 0;

	IF gSuperTrak.state.stateMachine.stateTransition.clear THEN

		IF NOT SumCritical THEN
			gSuperTrak.state.stateMachine.operationalState := CLEARING;

		ELSE
			Event_Code := 83;
			EventLog.Commands.WriteUserEvent := TRUE;
		END_IF;
	END_IF;
END_ACTION
```

#### Clearing.st
```iecst
ACTION Clearing:

		(*************************************************************************************************)
		(*************************************************************************************************)
		(* FUNCTION BLOCK CONFIGURATION *)

	Counter_Clearing_Timeout(IN := TRUE, PT := T#40s);

	(* Timer is connected to sensor variable and also to Target 4 so only hen a shuttle is at target 4 the time will start *)

	//If the clearing takes more time than expected the supertrak goes into aborted
	IF Counter_Clearing_Timeout.Q THEN
		Event_Code := 7;
		EventLog.Commands.WriteUserEvent := TRUE;
		gSuperTrak.state.stateMachine.stateTransition.abort := TRUE;
	END_IF;

	QA_Actuator_DOWN := TRUE;
	Timer_Actuator_DOWN (IN := TRUE, PT := T#8s);
	Outfeed_Actuator_DOWN := TRUE;
	Timer_Outfeed_DOWN (IN := TRUE, PT := T#30s);
	Outfeed_Actuator_BACK := TRUE;

	IF Timer_Actuator_DOWN.Q AND Timer_Outfeed_DOWN.Q THEN
		IF StControl_0.Active AND
			ST_LightBarrier_SecurityOut1_R AND ST_LightBarrier_SecurityOut2_R THEN

			(* Enable all sections for the calibration to begin *)
			CASE Calibration_State OF
				ENABLE_SYSTEM:
					//Assign to extarnal input for power enable
					StControl_0.EnableAllSections := TRUE;

					IF StControl_0.SectionsEnabled THEN
						FOR Index := 1 TO SUPERTRAK_TARGETS DO
							// Enable StTargetExt
							StTargetExt_[Index].Enable     := TRUE;
						END_FOR;

						Event_Code := 0;
						EventLog.Commands.WriteUserEvent := TRUE;

						(* Check if the calibration has been already done for the first time *)

						IF Last_ID = 0 THEN
							Counter_Clearing_Timeout(IN := FALSE);
							Calibration_State := ID_SETTING;
						ELSE
							Counter_Clearing_Timeout(IN := FALSE);
							Calibration_State := ABORTED_RESET_POSITIONS;
						END_IF;

						(* Variables initialization *)
						Calibration_Finished := FALSE;
						Shuttle := 0;
						Shuttle_sent := 0;
						New_ID := 0;
						First_ID := 0;
						first_shuttle := TRUE;
						Time_For_Stop(IN := FALSE, PT := T#3s);
					END_IF;

					(* Set id for each shuttle *)
				ID_SETTING:
					QA_Actuator_DOWN := FALSE;
					Outfeed_Actuator_DOWN := FALSE;
					Outfeed_Actuator_BACK := FALSE;

					(* If there is a shuttle at target 1 which id is 0 => No id given to that shuttle *)
					IF StTargetExt_[1].PalletPresent THEN
						(* Then the shuttle is given an id and sent to QA *)
						IF StTargetExt_[1].PalletID = 0 THEN
							New_ID := New_ID + 1;
							TargetControlParameters[1].PalletConfig.ID := New_ID;
							StTargetExt_[1].SetPalletID:= TRUE;
							Last_ID := New_ID;
							Calibration_State := SEND_TO_QA;

							(* When there are no more shuttles left and calibration has gone as it should *)
						ELSIF NOT StTargetExt_[4].PalletPresent AND Calibration_Finished THEN
							Calibration_State := CALIBRATION_END;
						END_IF;
					END_IF;

					(* If there is a shuttle at target 4 we take the ID and store the value in a variable, then release it to the parking *)
					IF StTargetExt_[4].PalletPresent THEN
						TargetControlParameters[1].AdvancedReleaseConfig.DestinationTarget  := 4;
						TargetControlParameters[4].AdvancedReleaseConfig.DestinationTarget  := 1;

						//If the shuttle at target 4 does not need to be checked it has to wait a certain time at target 4
						IF QA_finished THEN
							//Set timer to false each time we do something so the timer is not triggered
							Counter_Clearing_Timeout(IN := FALSE);

							StTargetExt_[4].ReleaseToTarget := TRUE;

							(* When we reach the last id at QA then we go to the last state of calibration *)
							IF StTargetExt_[4].PalletID = Last_ID THEN
								Calibration_Finished := TRUE;
							END_IF;

						END_IF;

					END_IF;

					(* When the shuttle leaves the target -> reset the ReleaseToTarget parameter*)
					IF EDGENEG(StTargetExt_[1].PalletPresent) THEN
						StTargetExt_[1].ReleaseToTarget := FALSE;
					END_IF;

					IF EDGENEG(StTargetExt_[4].PalletPresent) THEN
						StTargetExt_[4].ReleaseToTarget:= FALSE;
					END_IF;

					(* State for movement of shuttle when configured *)
				SEND_TO_QA:

					IF StTargetExt_[1].PalletID = 0 THEN
						TargetControlParameters[1].AdvancedReleaseConfig.MoveConfigIdx := 1;
						//Reset of SetPalletID so we can set the next one in ID_SETTING at Target 1
						StTargetExt_[1].SetPalletID:= FALSE;

					ELSE
						TargetControlParameters[1].AdvancedReleaseConfig.MoveConfigIdx := 1;
						TargetControlParameters[1].AdvancedReleaseConfig.DestinationTarget := 4;
						StTargetExt_[1].ReleaseToTarget := TRUE;

						Calibration_State := ID_SETTING;
					END_IF;

					(*************************************************)
					(* States for calibration from abort mid process*)
					(*************************************************)

					(* Send shuttles to target one after aborted *)
				ABORTED_RESET_POSITIONS:
					QA_Actuator_DOWN := FALSE;
					Outfeed_Actuator_BACK := FALSE;
					Outfeed_Actuator_DOWN := FALSE;

					(* In case there is a transition from aborted but calibration was already done we need to recalibrate and send the shuttle to QA *)
					IF transitionFromAborted AND (StTargetExt_[1].PalletID <> 0 OR (NOT StTargetExt_[1].PalletPresent AND Last_ID = SUPERTRAK_SHUTTLES)) THEN

						Time_For_AbortClearing_Start (IN := TRUE, PT := T#3s);

						(* Wait until we are sure every shuttle is not moving and near a target *)
						IF Time_For_AbortClearing_Start.Q THEN

							(* Timer long enough to be sure all shuttles are going to target 1*)
							Time_For_AbortClearing_End (IN := TRUE, PT := T#7s);

							(* Sending all shuttles to target one *)
							FOR j:= 1 TO SUPERTRAK_TARGETS DO
								//If there is a pallet present at a target
								IF StTargetExt_[j].PalletPresent THEN
									//Make sure the movement is the slow one
									TargetControlParameters[j].AdvancedReleaseConfig.MoveConfigIdx := 1;

									//If it is target eight
									IF j = 8 THEN
										IF first_shuttle THEN
											//Store the Id of first shuttle going to target one so we do not send it twice
											first_shuttle := FALSE;
											First_ID := StTargetExt_[j].PalletID;
										END_IF;
										//Final target is target 1 and the shuttle is released
										TargetControlParameters[j].AdvancedReleaseConfig.DestinationTarget := 1;
										gSuperTrak.skill.moveShuttle[StTargetExt_[j].PalletID].inputParameters.finalTarget := Target_1;
										//Setting the current target because the skills are in aborted so we need to set it beforehand
										gSuperTrak.skill.moveShuttle[StTargetExt_[j].PalletID].outputParameters.currentTarget := Target_1;
										StTargetExt_[8].ReleaseToTarget := TRUE;

										//Any other target releases it's shuttle to target 8
									ELSE
										TargetControlParameters[j].AdvancedReleaseConfig.DestinationTarget := 8;
									END_IF;

									(* Only release the shuttles one time *)
									IF j <> 1 OR StTargetExt_[1].PalletID <> First_ID THEN
										StTargetExt_[j].ReleaseToTarget := TRUE;
									END_IF;
								END_IF;

								//After the release has been done the parameter is reset
								IF StTargetExt_[j].CommandDone THEN
									StTargetExt_[j].ReleaseToTarget := FALSE;
								END_IF;

							END_FOR;
						END_IF;
					END_IF;

					IF Time_For_AbortClearing_End.Q THEN
						Counter_Clearing_Timeout(IN := FALSE);
						Counter_Check_Shuttle (IN := FALSE);
						Calibration_State := ABORTED_CALIBRATION;
					END_IF;

					(* Manual calibration and setup for the shuttles *)
				ABORTED_CALIBRATION:
					Time_For_AbortClearing_Start (IN := FALSE, PT := T#3s);
					Time_For_AbortClearing_End (IN := FALSE, PT := T#7s);

					(*In case some shuttles did not make it to target one we check the position 8 for them and release them to target 1*)
					IF StTargetExt_[8].PalletPresent AND NOT StTargetExt_[8].ReleaseToTarget THEN
						StTargetExt_[8].ReleaseToTarget := TRUE;
					END_IF;

					IF StTargetExt_[8].CommandDone THEN
						StTargetExt_[8].ReleaseToTarget := FALSE;
					END_IF;

					(* Set an ID to the Shuttle. If done for one of them should be done for all in order to avoid doubled IDs *)
					//This is not necessary to do
					//				IF SetID THEN
					//
					//					Counter_Clearing_Timeout(IN := FALSE);
					//
					//					New_ID := New_ID + 1;
					//					TargetControlParameters[1].PalletConfig.ID := New_ID;
					//					StTargetExt_[1].SetPalletID := TRUE;
					//					SetID := FALSE;

					(* Send shuttle to QA station *)
					IF StTargetExt_[1].PalletPresent AND Shuttle_sent < SUPERTRAK_SHUTTLES THEN
						Counter_Clearing_Timeout(IN := FALSE);
						Shuttle_sent := Shuttle_sent + 1;
						Calibration_State := ABORTED_SEND_TO_QA;
						//StTargetExt_[1].SetPalletID := FALSE;
					END_IF;

					(* Send shuttle to parking station *)
					IF QA_finished (*AND StTargetExt_[4].PalletPresent*) THEN

						(* Wheneer the release of the shuttle has been done the releasetotarget parameter is reset *)
						IF StTargetExt_[4].CommandDone THEN
							StTargetExt_[4].ReleaseToTarget := FALSE;

						ELSE
							TargetControlParameters[4].AdvancedReleaseConfig.MoveConfigIdx := 1;
							TargetControlParameters[4].AdvancedReleaseConfig.DestinationTarget  := 1;
							TargetControlParameters[4].AdvancedReleaseConfig.Direction     := stCOM_DIR_RIGHT;

							Shuttle := Shuttle + 1;

							Counter_Check_Shuttle(IN := FALSE);
							StTargetExt_[4].ReleaseToTarget := TRUE;
						END_IF;

						IF Shuttle_sent = Last_ID AND Shuttle = Last_ID THEN
							Calibration_Finished := TRUE;
						END_IF;

					END_IF;

					//				IF MES_Test THEN
					//					Calibration_State := CALIBRATION_END;
					//				END_IF;
					//

					IF StTargetExt_[1].CommandDone THEN
						StTargetExt_[1].ReleaseToTarget := FALSE;
					END_IF;

					IF Calibration_Finished THEN
						Calibration_State := CALIBRATION_END;
					END_IF;

				ABORTED_SEND_TO_QA:

					(* Sending shuttle to QA *)
					TargetControlParameters[1].AdvancedReleaseConfig.MoveConfigIdx := 1;
					TargetControlParameters[1].AdvancedReleaseConfig.DestinationTarget  := 4;
					TargetControlParameters[1].AdvancedReleaseConfig.Direction     := stCOM_DIR_RIGHT;

					StTargetExt_[1].ReleaseToTarget := TRUE;

					IF EDGENEG(StTargetExt_[1].PalletPresent) THEN
						StTargetExt_[1].SetPalletID := FALSE;
						Calibration_State := ABORTED_CALIBRATION;
					END_IF;

					(* Reconfiguration of process *)
				CALIBRATION_END:

					(* Activate the timer for the state machine to go in stop mode being sure the shuttle are not moving *)
					Time_For_Stop(IN := TRUE);

					(* Reconfigure the process routing and flow direction in case something was changed during calibration *)
					TargetControlParameters[1].AdvancedReleaseConfig.DestinationTarget  := 2;
					TargetControlParameters[1].AdvancedReleaseConfig.Direction     := stCOM_DIR_RIGHT;

					TargetControlParameters[2].AdvancedReleaseConfig.DestinationTarget  := 3;
					TargetControlParameters[2].AdvancedReleaseConfig.Direction     := stCOM_DIR_RIGHT;

					TargetControlParameters[3].AdvancedReleaseConfig.DestinationTarget  := 4;
					TargetControlParameters[3].AdvancedReleaseConfig.Direction     := stCOM_DIR_RIGHT;

					TargetControlParameters[4].AdvancedReleaseConfig.DestinationTarget  := 5;
					TargetControlParameters[4].AdvancedReleaseConfig.Direction     := stCOM_DIR_RIGHT;

					TargetControlParameters[5].AdvancedReleaseConfig.DestinationTarget  := 6;
					TargetControlParameters[5].AdvancedReleaseConfig.Direction     := stCOM_DIR_RIGHT;

					TargetControlParameters[6].AdvancedReleaseConfig.DestinationTarget  := 7;
					TargetControlParameters[6].AdvancedReleaseConfig.Direction     := stCOM_DIR_RIGHT;

					TargetControlParameters[7].AdvancedReleaseConfig.DestinationTarget  := 8;
					TargetControlParameters[7].AdvancedReleaseConfig.Direction     := stCOM_DIR_RIGHT;

					TargetControlParameters[8].AdvancedReleaseConfig.DestinationTarget  := 1;
					TargetControlParameters[8].AdvancedReleaseConfig.Direction     := stCOM_DIR_RIGHT;

					IF Time_For_Stop.Q THEN
						//Disable the timer until we get to clearing again
						Counter_Clearing_Timeout(IN := FALSE);
						gSuperTrak.state.stateMachine.operationalState := STOPPED;
					END_IF;
			END_CASE;
		END_IF;
	END_IF;
END_ACTION
```

#### Stopped.st
```iecst
ACTION Stopped:

	QA_Actuator_DOWN := FALSE;
	Timer_Actuator_DOWN (IN := FALSE);
	Outfeed_Actuator_DOWN := FALSE;
	Timer_Outfeed_DOWN (IN := FALSE);
	Outfeed_Actuator_BACK := FALSE;

	IF	gSuperTrak.state.stateMachine.stateTransition.reset THEN
		gSuperTrak.state.stateMachine.operationalState := RESETTING;
	END_IF;

END_ACTION
```

#### Stopping.st
```iecst
ACTION Stopping:

	// Loop thru all StTargetExt function blocks
	FOR j := 1 TO SUPERTRAK_TARGETS DO
		// Enable StTargetExt
		StTargetExt_[j].ReleaseToTarget		:= FALSE;
	END_FOR;

	Transition_From_Stopped := TRUE;

	Skills_Aborted := 0;

	//Send abort transition to the skills
	gSuperTrak.skill.checkParking.state.stateMachine.stateTransition.abort := TRUE;

	FOR iShuttle := 1 TO SUPERTRAK_SHUTTLES DO
		gSuperTrak.skill.moveShuttle[iShuttle].state.stateMachine.stateTransition.abort := TRUE;
	END_FOR;

	gSuperTrak.state.stateMachine.operationalState := STOPPED;

END_ACTION
```

#### Holding.st
```iecst
ACTION Holding:

	gSuperTrak.state.stateMachine.operationalState := HELD;

END_ACTION
```

#### Held.st
```iecst
ACTION Held:

	IF NOT Outfeed_Full THEN

		TON_Restore_Outfeed(IN := TRUE, PT := T#10s);

		IF TON_Restore_Outfeed.Q THEN

			Event_Code := 81;
			EventLog.Commands.WriteUserEvent := TRUE;

		END_IF;

	END_IF;

	IF gSuperTrak.state.stateMachine.stateTransition.unhold THEN
		TON_Restore_Outfeed(IN := FALSE);
		gSuperTrak.state.stateMachine.operationalState := UNHOLDING;

	END_IF;

END_ACTION
```

#### Unholding.st
```iecst
ACTION Unholding:

	gSuperTrak.state.stateMachine.operationalState := RUNNING;

END_ACTION
```

#### Running.st
```iecst
ACTION Running:

	(* For each of the skills we check if there is an STOPPED state *)
	FOR j := 1 TO SUPERTRAK_SHUTTLES DO
		IF gSuperTrak.skill.moveShuttle[j].state.stateMachine.operationalState = STOPPED THEN

			Timer_Send_Super_Trak_In_Stop(IN := TRUE, PT := T#2s);

			IF Timer_Send_Super_Trak_In_Stop.Q = TRUE THEN
				Timer_Send_Super_Trak_In_Stop(IN := FALSE);

				Event_Code := 82;
				EventLog.Commands.WriteUserEvent := TRUE;

				gSuperTrak.state.stateMachine.stateTransition.stop := TRUE;

			END_IF;
		END_IF;
	END_FOR;

	(* If not we wait for the pause trigger *)
	IF	gSuperTrak.state.stateMachine.stateTransition.pause THEN
		gSuperTrak.state.stateMachine.operationalState := PAUSING;
	END_IF;

	Timer_Send_Super_Trak_In_Stop();
END_ACTION
```

#### Suspending.st
```iecst
ACTION Suspending:

	gSuperTrak.state.stateMachine.operationalState := SUSPENDED;

END_ACTION
```

#### Paused.st
```iecst
ACTION Paused:

	IF gSuperTrak.state.stateMachine.stateTransition.resume THEN
		gSuperTrak.state.stateMachine.operationalState := RUNNING;

	END_IF;

END_ACTION
```

#### Unsuspending.st
```iecst
ACTION Unsuspending:

	IF gSuperTrak.state.stateMachine.stateTransition.suspend THEN
		gSuperTrak.state.stateMachine.operationalState := SUSPENDING;
	ELSE
		gSuperTrak.state.stateMachine.operationalState := RUNNING;
	END_IF;

END_ACTION
```

#### Complete.st
```iecst
ACTION Complete:

	IF gSuperTrak.state.stateMachine.stateTransition.reset THEN
		gSuperTrak.state.stateMachine.operationalState := RESETTING;

	END_IF;

END_ACTION
```

#### moveShuttle.st
```iecst
ACTION moveShuttle:
		(*************************************************************************************************)
		(*************************************************************************************************)
		(* State Machine *)
	CASE gSuperTrak.skill.moveShuttle[iShuttle].state.stateMachine.operationalState OF
		(*************************************************************************************************)
		(* RESETTING *)
		RESETTING:
			(*gSuperTrak.skill.moveShuttle[iShuttle].state.stateMachine.stateTransition.reset := FALSE;*)

			IF gSuperTrak.skill.moveShuttle[iShuttle].state.stateMachine.stateTransition.abort THEN
				gSuperTrak.skill.moveShuttle[iShuttle].state.stateMachine.operationalState := ABORTING;

			ELSIF gSuperTrak.skill.moveShuttle[iShuttle].state.stateMachine.stateTransition.stop THEN
				gSuperTrak.skill.moveShuttle[iShuttle].state.stateMachine.operationalState := STOPPING;

			ELSE
				moveShuttle_Resetting;

			END_IF;

			(*************************************************************************************************)
			(* IDLE *)
		IDLE:
			gSuperTrak.skill.moveShuttle[iShuttle].state.stateMachine.stateTransition.reset := FALSE;

			IF gSuperTrak.skill.moveShuttle[iShuttle].state.stateMachine.stateTransition.abort THEN
				gSuperTrak.skill.moveShuttle[iShuttle].state.stateMachine.operationalState := ABORTING;

			ELSIF gSuperTrak.skill.moveShuttle[iShuttle].state.stateMachine.stateTransition.stop THEN
				gSuperTrak.skill.moveShuttle[iShuttle].state.stateMachine.operationalState := STOPPING;

			ELSE
				moveShuttle_Idle;

			END_IF;

			(*************************************************************************************************)
			(* STARTING *)
		STARTING:
			//			gSuperTrak.skill.moveShuttle[iShuttle].state.stateMachine.stateTransition.start := FALSE;

			IF gSuperTrak.skill.moveShuttle[iShuttle].state.stateMachine.stateTransition.abort THEN
				gSuperTrak.skill.moveShuttle[iShuttle].state.stateMachine.operationalState := ABORTING;

			ELSIF gSuperTrak.skill.moveShuttle[iShuttle].state.stateMachine.stateTransition.stop THEN
				gSuperTrak.skill.moveShuttle[iShuttle].state.stateMachine.operationalState := STOPPING;

			ELSE
				moveShuttle_Starting;

			END_IF;

			(*************************************************************************************************)
			(* RUNNING *)
		RUNNING:

			gSuperTrak.skill.moveShuttle[iShuttle].state.stateMachine.stateTransition.start := FALSE;

			IF gSuperTrak.skill.moveShuttle[iShuttle].state.stateMachine.stateTransition.abort THEN
				gSuperTrak.skill.moveShuttle[iShuttle].state.stateMachine.operationalState := ABORTING;

			ELSIF gSuperTrak.skill.moveShuttle[iShuttle].state.stateMachine.stateTransition.stop THEN
				gSuperTrak.skill.moveShuttle[iShuttle].state.stateMachine.operationalState := STOPPING;

			ELSIF gSuperTrak.skill.moveShuttle[iShuttle].state.stateMachine.stateTransition.hold THEN

				//				gSuperTrak.skill.moveShuttle[iShuttle].state.stateMachine.operationalState := HOLDING;

			ELSIF gSuperTrak.skill.moveShuttle[iShuttle].state.stateMachine.stateTransition.suspend THEN

				//				gSuperTrak.skill.moveShuttle[iShuttle].state.stateMachine.operationalState := SUSPENDING;

			ELSIF gSuperTrak.skill.moveShuttle[iShuttle].state.stateMachine.stateTransition.pause THEN

				//				gSuperTrak.skill.moveShuttle[iShuttle].state.stateMachine.operationalState := PAUSING;

			ELSE
				moveShuttle_Running;

			END_IF;

			(*************************************************************************************************)
			(* PAUSING *)
		PAUSING:
			(*gSuperTrak.skill.moveShuttle[iShuttle].state.stateMachine.stateTransition.pause := FALSE;*)

			IF gSuperTrak.skill.moveShuttle[iShuttle].state.stateMachine.stateTransition.abort THEN
				gSuperTrak.skill.moveShuttle[iShuttle].state.stateMachine.operationalState := ABORTING;

			ELSIF gSuperTrak.skill.moveShuttle[iShuttle].state.stateMachine.stateTransition.stop THEN
				gSuperTrak.skill.moveShuttle[iShuttle].state.stateMachine.operationalState := STOPPING;

			ELSIF gSuperTrak.skill.moveShuttle[iShuttle].state.stateMachine.stateTransition.hold THEN

				//				gSuperTrak.skill.moveShuttle[iShuttle].state.stateMachine.operationalState := HOLDING;

			ELSIF gSuperTrak.skill.moveShuttle[iShuttle].state.stateMachine.stateTransition.suspend THEN

				//				gSuperTrak.skill.moveShuttle[iShuttle].state.stateMachine.operationalState := SUSPENDING;

			ELSE
				moveShuttle_Pausing;
			END_IF;

			(*************************************************************************************************)
			(* PAUSED *)
		PAUSED:

			gSuperTrak.skill.moveShuttle[iShuttle].state.stateMachine.stateTransition.pause := FALSE;

			IF gSuperTrak.skill.moveShuttle[iShuttle].state.stateMachine.stateTransition.abort THEN
				gSuperTrak.skill.moveShuttle[iShuttle].state.stateMachine.operationalState := ABORTING;

			ELSIF gSuperTrak.skill.moveShuttle[iShuttle].state.stateMachine.stateTransition.stop THEN
				gSuperTrak.skill.moveShuttle[iShuttle].state.stateMachine.operationalState := STOPPING;

			ELSIF gSuperTrak.skill.moveShuttle[iShuttle].state.stateMachine.stateTransition.hold THEN

				//				gSuperTrak.skill.moveShuttle[iShuttle].state.stateMachine.operationalState := HOLDING;

			ELSIF gSuperTrak.skill.moveShuttle[iShuttle].state.stateMachine.stateTransition.suspend THEN

				//				gSuperTrak.skill.moveShuttle[iShuttle].state.stateMachine.operationalState := SUSPENDING;

			ELSE
				moveShuttle_Paused;

			END_IF;

			(*************************************************************************************************)
			(* SUSPENDING *)
		SUSPENDING:
			(*gSuperTrak.skill.moveShuttle[iShuttle].state.stateMachine.stateTransition.suspend := FALSE;*)

			IF gSuperTrak.skill.moveShuttle[iShuttle].state.stateMachine.stateTransition.abort THEN
				gSuperTrak.skill.moveShuttle[iShuttle].state.stateMachine.operationalState := ABORTING;

			ELSIF gSuperTrak.skill.moveShuttle[iShuttle].state.stateMachine.stateTransition.stop THEN
				gSuperTrak.skill.moveShuttle[iShuttle].state.stateMachine.operationalState := STOPPING;

			ELSIF gSuperTrak.skill.moveShuttle[iShuttle].state.stateMachine.stateTransition.hold THEN

				//				gSuperTrak.skill.moveShuttle[iShuttle].state.stateMachine.operationalState := HOLDING;

			ELSE
				moveShuttle_Suspending;

			END_IF;

			(*************************************************************************************************)
			(* SUSPENDED *)
		SUSPENDED:

			gSuperTrak.skill.moveShuttle[iShuttle].state.stateMachine.stateTransition.suspend := FALSE;

			IF gSuperTrak.skill.moveShuttle[iShuttle].state.stateMachine.stateTransition.abort THEN
				gSuperTrak.skill.moveShuttle[iShuttle].state.stateMachine.operationalState := ABORTING;

			ELSIF gSuperTrak.skill.moveShuttle[iShuttle].state.stateMachine.stateTransition.stop THEN
				gSuperTrak.skill.moveShuttle[iShuttle].state.stateMachine.operationalState := STOPPING;

			ELSIF gSuperTrak.skill.moveShuttle[iShuttle].state.stateMachine.stateTransition.hold THEN

				//				gSuperTrak.skill.moveShuttle[iShuttle].state.stateMachine.operationalState := HOLDING;

			ELSE
				moveShuttle_Suspended;

			END_IF;

			(*************************************************************************************************)
			(* UNSUSPENDING *)
		UNSUSPENDING:
			gSuperTrak.skill.moveShuttle[iShuttle].state.stateMachine.stateTransition.unsuspend := FALSE;

			IF gSuperTrak.skill.moveShuttle[iShuttle].state.stateMachine.stateTransition.abort THEN
				gSuperTrak.skill.moveShuttle[iShuttle].state.stateMachine.operationalState := ABORTING;

			ELSIF gSuperTrak.skill.moveShuttle[iShuttle].state.stateMachine.stateTransition.stop THEN
				gSuperTrak.skill.moveShuttle[iShuttle].state.stateMachine.operationalState := STOPPING;

			ELSIF gSuperTrak.skill.moveShuttle[iShuttle].state.stateMachine.stateTransition.hold THEN

				//				gSuperTrak.skill.moveShuttle[iShuttle].state.stateMachine.operationalState := HOLDING;

			ELSE
				moveShuttle_Unsuspending;

			END_IF;

			(*************************************************************************************************)
			(* HOLDING *)
		HOLDING:
			(*gSuperTrak.skill.moveShuttle[iShuttle].state.stateMachine.stateTransition.hold := FALSE;*)

			IF gSuperTrak.skill.moveShuttle[iShuttle].state.stateMachine.stateTransition.abort THEN
				gSuperTrak.skill.moveShuttle[iShuttle].state.stateMachine.operationalState := ABORTING;

			ELSIF gSuperTrak.skill.moveShuttle[iShuttle].state.stateMachine.stateTransition.stop THEN
				gSuperTrak.skill.moveShuttle[iShuttle].state.stateMachine.operationalState := STOPPING;

			ELSE
				moveShuttle_Holding;

			END_IF;

			(*************************************************************************************************)
			(* HELD *)
		HELD:

			gSuperTrak.skill.moveShuttle[iShuttle].state.stateMachine.stateTransition.hold := FALSE;

			IF gSuperTrak.skill.moveShuttle[iShuttle].state.stateMachine.stateTransition.abort THEN
				gSuperTrak.skill.moveShuttle[iShuttle].state.stateMachine.operationalState := ABORTING;

			ELSIF gSuperTrak.skill.moveShuttle[iShuttle].state.stateMachine.stateTransition.stop THEN
				gSuperTrak.skill.moveShuttle[iShuttle].state.stateMachine.operationalState := STOPPING;

			ELSE
				moveShuttle_Held;

			END_IF;

			(*************************************************************************************************)
			(* UNHOLDING *)
		UNHOLDING:
			gSuperTrak.skill.moveShuttle[iShuttle].state.stateMachine.stateTransition.unhold := FALSE;

			IF gSuperTrak.skill.moveShuttle[iShuttle].state.stateMachine.stateTransition.abort THEN
				gSuperTrak.skill.moveShuttle[iShuttle].state.stateMachine.operationalState := ABORTING;

			ELSIF gSuperTrak.skill.moveShuttle[iShuttle].state.stateMachine.stateTransition.stop THEN
				gSuperTrak.skill.moveShuttle[iShuttle].state.stateMachine.operationalState := STOPPING;

			ELSE
				moveShuttle_Unholding;

			END_IF;

			(*************************************************************************************************)
			(* COMPLETING *)
		COMPLETING:

			IF gSuperTrak.skill.moveShuttle[iShuttle].state.stateMachine.stateTransition.abort THEN
				gSuperTrak.skill.moveShuttle[iShuttle].state.stateMachine.operationalState := ABORTING;

			ELSIF gSuperTrak.skill.moveShuttle[iShuttle].state.stateMachine.stateTransition.stop THEN
				gSuperTrak.skill.moveShuttle[iShuttle].state.stateMachine.operationalState := STOPPING;

			ELSE
				moveShuttle_Completing;

			END_IF;

			(*************************************************************************************************)
			(* COMPLETE *)
		COMPLETE:

			IF gSuperTrak.skill.moveShuttle[iShuttle].state.stateMachine.stateTransition.abort THEN
				gSuperTrak.skill.moveShuttle[iShuttle].state.stateMachine.operationalState := ABORTING;

			ELSIF gSuperTrak.skill.moveShuttle[iShuttle].state.stateMachine.stateTransition.stop THEN
				gSuperTrak.skill.moveShuttle[iShuttle].state.stateMachine.operationalState := STOPPING;

			ELSE
				moveShuttle_Complete;

			END_IF;

			(*************************************************************************************************)
			(* STOPPING *)
		STOPPING:
			//			gSuperTrak.skill.moveShuttle[iShuttle].state.stateMachine.stateTransition.stop := FALSE;

			IF gSuperTrak.skill.moveShuttle[iShuttle].state.stateMachine.stateTransition.abort THEN
				gSuperTrak.skill.moveShuttle[iShuttle].state.stateMachine.operationalState := ABORTING;

			ELSE
				moveShuttle_Stopping;

			END_IF;

			(*************************************************************************************************)
			(* STOPPED *)
		STOPPED:

			gSuperTrak.skill.moveShuttle[iShuttle].state.stateMachine.stateTransition.stop := FALSE;

			IF gSuperTrak.skill.moveShuttle[iShuttle].state.stateMachine.stateTransition.abort THEN
				gSuperTrak.skill.moveShuttle[iShuttle].state.stateMachine.operationalState := ABORTING;

			ELSE
				moveShuttle_Stopped;

			END_IF;

			(*************************************************************************************************)
			(* ABORTING *)
		ABORTING:
			(*gSuperTrak.skill.moveShuttle[iShuttle].state.stateMachine.stateTransition.abort := FALSE;*)

			moveShuttle_Aborting;

			(*************************************************************************************************)
			(* ABORTED *)
		ABORTED:

			gSuperTrak.skill.moveShuttle[iShuttle].state.stateMachine.stateTransition.abort := FALSE;

			moveShuttle_Aborted;

			(*************************************************************************************************)
			(* CLEARING *)
		CLEARING:
			gSuperTrak.skill.moveShuttle[iShuttle].state.stateMachine.stateTransition.clear := FALSE;

			moveShuttle_Clearing;

			(*************************************************************************************************)
			(* ELSE *)
		ELSE;

	END_CASE;
END_ACTION
```

#### Program Logical/SuperTrak_Module/StateMachine_SuperTrak/moveShuttle/StateActions

##### moveShuttle_Aborted.st
```iecst
ACTION moveShuttle_Aborted:

	IF gSuperTrak.skill.moveShuttle[iShuttle].state.stateMachine.stateTransition.reset THEN
		gSuperTrak.skill.moveShuttle[iShuttle].state.stateMachine.operationalState := RESETTING;

	ELSIF gSuperTrak.skill.moveShuttle[iShuttle].state.stateMachine.stateTransition.clear THEN
		gSuperTrak.skill.moveShuttle[iShuttle].state.stateMachine.operationalState := CLEARING;

	END_IF;

END_ACTION
```

##### moveShuttle_Aborting.st
```iecst
ACTION moveShuttle_Aborting:
//
//	IF NOT Transition_From_Stopped AND gSuperTrak.state.stateMachine.operationalState <> ABORTING THEN
//		Event_Code := iShuttle + 65;
//		EventLog.Commands.WriteUserEvent := TRUE;
//	END_IF;

	//Not knowing if any trigger was set to true before the abort we make sure every one of them is false before going to aborted
	gSuperTrak.skill.moveShuttle[iShuttle].state.stateMachine.stateTransition.abort 	:= FALSE;
	gSuperTrak.skill.moveShuttle[iShuttle].state.stateMachine.stateTransition.clear 	:= FALSE;
	gSuperTrak.skill.moveShuttle[iShuttle].state.stateMachine.stateTransition.hold 		:= FALSE;
	gSuperTrak.skill.moveShuttle[iShuttle].state.stateMachine.stateTransition.pause 	:= FALSE;
	gSuperTrak.skill.moveShuttle[iShuttle].state.stateMachine.stateTransition.reset 	:= FALSE;
	gSuperTrak.skill.moveShuttle[iShuttle].state.stateMachine.stateTransition.resume 	:= FALSE;
	gSuperTrak.skill.moveShuttle[iShuttle].state.stateMachine.stateTransition.start 	:= FALSE;
	gSuperTrak.skill.moveShuttle[iShuttle].state.stateMachine.stateTransition.stop 		:= FALSE;
	gSuperTrak.skill.moveShuttle[iShuttle].state.stateMachine.stateTransition.suspend 	:= FALSE;
	gSuperTrak.skill.moveShuttle[iShuttle].state.stateMachine.stateTransition.unhold 	:= FALSE;
	gSuperTrak.skill.moveShuttle[iShuttle].state.stateMachine.stateTransition.unsuspend := FALSE;

	Skills_Aborted := Skills_Aborted + 1;
	gSuperTrak.skill.moveShuttle[iShuttle].state.stateMachine.operationalState := ABORTED;

END_ACTION
```

##### moveShuttle_Clearing.st
```iecst
ACTION moveShuttle_Clearing:

	gSuperTrak.skill.moveShuttle[iShuttle].state.stateMachine.stateTransition.clear := FALSE;

	gSuperTrak.skill.moveShuttle[iShuttle].state.stateMachine.operationalState := STOPPED;

END_ACTION
```

##### moveShuttle_Held.st
```iecst
ACTION moveShuttle_Held:

	IF gSuperTrak.skill.moveShuttle[iShuttle].state.stateMachine.stateTransition.unhold THEN
		gSuperTrak.skill.moveShuttle[iShuttle].state.stateMachine.operationalState := UNHOLDING;
	END_IF;

END_ACTION
```

##### moveShuttle_Holding.st
```iecst
ACTION moveShuttle_Holding:

	gSuperTrak.skill.moveShuttle[iShuttle].state.stateMachine.operationalState := HELD;

END_ACTION
```

##### moveShuttle_Pausing.st
```iecst
ACTION moveShuttle_Pausing:

	gSuperTrak.skill.moveShuttle[iShuttle].state.stateMachine.operationalState := PAUSED;

END_ACTION
```

##### moveShuttle_Resetting.st
```iecst
ACTION moveShuttle_Resetting:

	gSuperTrak.skill.moveShuttle[iShuttle].state.stateMachine.operationalState := IDLE;

END_ACTION
```

##### moveShuttle_Running.st
```iecst
ACTION moveShuttle_Running:
(* SuperTrak searchs for Shuttles at each target, and if it has arrived to the destination then we update the current target and
	the skill jumps	into completing *)

	FOR i[iShuttle] := 1 TO SUPERTRAK_TARGETS DO

		//In case there was an error and the release to target parameter is not set we set it and retry
//		IF StTargetExt_[i[iShuttle]].PalletPresent AND
//			StTargetExt_[i[iShuttle]].PalletID = iShuttle AND
//			gSuperTrak.skill.moveShuttle[iShuttle].outputParameters.currentTarget = i[iShuttle] THEN
//
//			IF NOT StTargetExt_[i[iShuttle]].ReleaseToTarget THEN
//				StTargetExt_[i[iShuttle]].ReleaseToTarget := TRUE;
//			END_IF;
//
//		END_IF;

		//If the shuttle reaches destination
		IF StTargetExt_[i[iShuttle]].PalletPresent AND
			StTargetExt_[i[iShuttle]].PalletID = iShuttle AND
			gSuperTrak.skill.moveShuttle[iShuttle].inputParameters.finalTarget = USINT_TO_UDINT(i[iShuttle]) THEN

			IF gSuperTrak.skill.moveShuttle[iShuttle].inputParameters.finalTarget = 8
				AND gSuperTrak.skill.moveShuttle[iShuttle].outputParameters.currentTarget = 7
				AND Set_Info_Messages THEN

				Event_Code := 41 + iShuttle;
				EventLog.Commands.WriteUserEvent := TRUE;

			END_IF;

			gSuperTrak.skill.moveShuttle[iShuttle].outputParameters.currentTarget := i[iShuttle];
			gSuperTrak.skill.moveShuttle[iShuttle].state.stateMachine.operationalState := COMPLETING;

		END_IF;

	END_FOR;
END_ACTION
```

##### moveShuttle_Starting.st
```iecst
ACTION moveShuttle_Starting:

	(* ************************************************************************** *)
	(* starting move skill if pallet is in queueing infront of Target_8 *)

	IF	(gSuperTrak.skill.moveShuttle[iShuttle].outputParameters.currentTarget = Target_8 AND
		gSuperTrak.skill.moveShuttle[iShuttle].inputParameters.finalTarget = Target_1) THEN

		gSuperTrak.skill.moveShuttle[iShuttle].state.stateMachine.stateTransition.start := FALSE;
		gSuperTrak.skill.moveShuttle[iShuttle].state.stateMachine.operationalState := RUNNING;

	END_IF;

	// Set Destination Target and direction of the Shuttle, Release shuttle to Target

FOR i[iShuttle] := 1 TO SUPERTRAK_TARGETS DO
			(* If there is a shuttle present at the target, which ID is the one MES wants to release,
		 and it's final target is not the target it is at, then we configure the movement and execute the release of the shuttle from the target *)
		IF StTargetExt_[i[iShuttle]].PalletPresent AND
			StTargetExt_[i[iShuttle]].PalletID = iShuttle AND
			gSuperTrak.skill.moveShuttle[iShuttle].inputParameters.finalTarget <> USINT_TO_UDINT(i[iShuttle]) THEN

			TargetControlParameters[i[iShuttle]].AdvancedReleaseConfig.DestinationTarget		:= UDINT_TO_USINT(gSuperTrak.skill.moveShuttle[iShuttle].inputParameters.finalTarget);
			TargetControlParameters[i[iShuttle]].AdvancedReleaseConfig.Direction				:= stCOM_DIR_RIGHT;

			(* If the final target is virtual target 8 or parking, the movement is set to be fast
			otherwise the movement will be slower because of the loaded shuttle *)
			IF TargetControlParameters[i[iShuttle]].AdvancedReleaseConfig.DestinationTarget = 1 OR
				TargetControlParameters[i[iShuttle]].AdvancedReleaseConfig.DestinationTarget = 8 THEN

				//Fast movement (See movement profiles in TrakMaster)
				TargetControlParameters[i[iShuttle]].AdvancedReleaseConfig.MoveConfigIdx := 2;

			ELSE
				//Slow movement (See movement profiles in TrakMaster)
				TargetControlParameters[i[iShuttle]].AdvancedReleaseConfig.MoveConfigIdx := 1;

			END_IF;

			IF StTargetExt_[i[iShuttle]].ReleaseToTarget  AND StTargetExt_[i[iShuttle]].CommandDone THEN
				StTargetExt_[i[iShuttle]].ReleaseToTarget := FALSE;

			ELSE
				StTargetExt_[i[iShuttle]].ReleaseToTarget := TRUE;
				(* After release skill goes into running state *)
				gSuperTrak.skill.moveShuttle[iShuttle].state.stateMachine.operationalState := RUNNING;
			END_IF;

		END_IF;

END_FOR;

END_ACTION
```

##### moveShuttle_Stopping.st
```iecst
ACTION moveShuttle_Stopping:
	(* Updates all the shuttles current target before entering stopped state *)
	FOR i[iShuttle] := 1 TO SUPERTRAK_TARGETS DO
		IF StTargetExt_[i[iShuttle]].PalletPresent AND
			StTargetExt_[i[iShuttle]].PalletID = iShuttle AND
			gSuperTrak.skill.moveShuttle[iShuttle].inputParameters.finalTarget = USINT_TO_UDINT(i[iShuttle]) THEN

			gSuperTrak.skill.moveShuttle[iShuttle].outputParameters.currentTarget := i[iShuttle];
			gSuperTrak.skill.moveShuttle[iShuttle].state.stateMachine.operationalState := STOPPED;
		END_IF;
	END_FOR;

	gSuperTrak.skill.moveShuttle[iShuttle].state.stateMachine.operationalState := STOPPED;
END_ACTION
```

##### moveShuttle_Suspended.st
```iecst
ACTION moveShuttle_Suspended:

	IF gSuperTrak.skill.moveShuttle[iShuttle].state.stateMachine.stateTransition.unsuspend THEN
		gSuperTrak.skill.moveShuttle[iShuttle].state.stateMachine.operationalState := UNSUSPENDING;
	END_IF;

END_ACTION
```

##### moveShuttle_Suspending.st
```iecst
ACTION moveShuttle_Suspending:

	gSuperTrak.skill.moveShuttle[iShuttle].state.stateMachine.operationalState := SUSPENDED;

END_ACTION
```

##### moveShuttle_Unholding.st
```iecst
ACTION moveShuttle_Unholding:

		gSuperTrak.skill.moveShuttle[iShuttle].state.stateMachine.operationalState := RUNNING;

END_ACTION
```

#### checkParking_Aborting.st
```iecst
ACTION checkParking_Aborting:

//	IF NOT Transition_From_Stopped AND gSuperTrak.state.stateMachine.operationalState <> ABORTING THEN
//		Event_Code := 77;
//		EventLog.Commands.WriteUserEvent := TRUE;
//	END_IF;
//

	//Not knowing if any trigger was set to true before the abort we make sure every one of them is false before going to aborted
	gSuperTrak.skill.checkParking.state.stateMachine.stateTransition.abort 		:= FALSE;
	gSuperTrak.skill.checkParking.state.stateMachine.stateTransition.clear 		:= FALSE;
	gSuperTrak.skill.checkParking.state.stateMachine.stateTransition.hold 		:= FALSE;
	gSuperTrak.skill.checkParking.state.stateMachine.stateTransition.pause 		:= FALSE;
	gSuperTrak.skill.checkParking.state.stateMachine.stateTransition.reset 		:= FALSE;
	gSuperTrak.skill.checkParking.state.stateMachine.stateTransition.resume 	:= FALSE;
	gSuperTrak.skill.checkParking.state.stateMachine.stateTransition.start 		:= FALSE;
	gSuperTrak.skill.checkParking.state.stateMachine.stateTransition.stop 		:= FALSE;
	gSuperTrak.skill.checkParking.state.stateMachine.stateTransition.suspend 	:= FALSE;
	gSuperTrak.skill.checkParking.state.stateMachine.stateTransition.unhold 	:= FALSE;
	gSuperTrak.skill.checkParking.state.stateMachine.stateTransition.unsuspend 	:= FALSE;

	Skills_Aborted := Skills_Aborted + 1;
	gSuperTrak.skill.checkParking.state.stateMachine.operationalState := ABORTED;

END_ACTION
```

#### checkParking_Stopped.st
```iecst
ACTION checkParking_Stopped:

	IF gSuperTrak.skill.checkParking.state.stateMachine.stateTransition.reset
	(*AND	NOT gbMessageSumAlarm*) THEN

		gSuperTrak.skill.checkParking.state.stateMachine.operationalState := RESETTING;
	END_IF;

END_ACTION
```

#### checkParking_Idle.st
```iecst
ACTION checkParking_Idle:

	IF gSuperTrak.skill.checkParking.state.stateMachine.stateTransition.start THEN

		gSuperTrak.skill.checkParking.state.stateMachine.operationalState := STARTING;

	END_IF

END_ACTION
```

#### checkParking_Resetting.st
```iecst
ACTION checkParking_Resetting:
	(* Alarm message?? *)

	gSuperTrak.skill.checkParking.state.stateMachine.operationalState := IDLE;
END_ACTION
```

#### checkParking_Holding.st
```iecst
ACTION checkParking_Holding:

	gSuperTrak.skill.checkParking.state.stateMachine.operationalState := HELD;

END_ACTION
```

#### checkParking_Held.st
```iecst
ACTION checkParking_Held:

	IF gSuperTrak.skill.checkParking.state.stateMachine.stateTransition.unhold THEN
		gSuperTrak.skill.checkParking.state.stateMachine.operationalState := UNHOLDING;
	END_IF;

END_ACTION
```

#### checkParking_Suspended.st
```iecst
ACTION checkParking_Suspended:

	IF gSuperTrak.skill.checkParking.state.stateMachine.stateTransition.unsuspend THEN
		gSuperTrak.skill.checkParking.state.stateMachine.operationalState := UNSUSPENDING;
	END_IF;

END_ACTION
```

#### checkParking_Paused.st
```iecst
ACTION checkParking_Paused:

	IF gSuperTrak.skill.checkParking.state.stateMachine.stateTransition.resume THEN
		gSuperTrak.skill.checkParking.state.stateMachine.operationalState := RUNNING;

	END_IF;

END_ACTION
```

#### checkParking_Running.st
```iecst
ACTION checkParking_Running:

//	FOR j := 1 TO 6 DO
//
//		IF gSuperTrak.skill.moveShuttle[j].outputParameters.currentTarget = 1 AND
//			 gSuperTrak.skill.moveShuttle[j].inputParameters.finalTarget = 8 THEN
//
//
//			shuttleCounter := shuttleCounter + 1;
//
//		END_IF;
//
//		IF shuttleCounter = 1 THEN
//
//			Last_Shuttle := -1;
//
//		END_IF;
//
//	END_FOR;
//
//	shuttleCounter := 0;

	(* If there is a Shuttle at parking position the supertrak reads and returns the ID to the MES,
	if there is no shuttle the returned value is -1 *)

	IF StTargetExt_[1].PalletPresent AND Last_Shuttle <> StTargetExt_[1].PalletID THEN
		gSuperTrak.skill.checkParking.outputParameters.shuttleId := StTargetExt_[1].PalletID;
		Last_Shuttle := StTargetExt_[1].PalletID;
		//		check_Parking_Timeout(IN := FALSE, PT:= T#5s);
	ELSE
		gSuperTrak.skill.checkParking.outputParameters.shuttleId  := -1;
//		check_Parking_Timeout(IN := TRUE, PT:= T#5s);

	END_IF;

	(* If we timeout then the las shuttle is forgotten *)
//	IF check_Parking_Timeout.Q THEN
//		Last_Shuttle := 0;
//	END_IF;

	(* After that Skill goes into completing state *)
	gSuperTrak.skill.checkParking.state.stateMachine.operationalState := COMPLETING;

END_ACTION
```

#### Outfeed.st
```iecst
ACTION Outfeed:
		(*************************************************************************************************)
		(*************************************************************************************************)
		(* State Machine *)
	CASE gSuperTrak.skill.Outfeed.state.stateMachine.operationalState OF
		(*************************************************************************************************)
		(* RESETTING *)
		RESETTING:
			(*gSuperTrak.skill.Outfeed.state.stateMachine.stateTransition.reset := FALSE;*)

			IF gSuperTrak.skill.Outfeed.state.stateMachine.stateTransition.abort THEN
				gSuperTrak.skill.Outfeed.state.stateMachine.operationalState := ABORTING;

			ELSIF gSuperTrak.skill.Outfeed.state.stateMachine.stateTransition.stop THEN
				gSuperTrak.skill.Outfeed.state.stateMachine.operationalState := STOPPING;

			ELSE
				Outfeed_Resetting;

			END_IF;

		(*************************************************************************************************)
		(* IDLE *)
		IDLE:
			gSuperTrak.skill.Outfeed.state.stateMachine.stateTransition.reset := FALSE;

			IF gSuperTrak.skill.Outfeed.state.stateMachine.stateTransition.abort THEN
				gSuperTrak.skill.Outfeed.state.stateMachine.operationalState := ABORTING;

			ELSIF gSuperTrak.skill.Outfeed.state.stateMachine.stateTransition.stop THEN
				gSuperTrak.skill.Outfeed.state.stateMachine.operationalState := STOPPING;

			ELSE
				Outfeed_Idle;

			END_IF;

		(*************************************************************************************************)
		(* STARTING *)
		STARTING:

			IF gSuperTrak.skill.Outfeed.state.stateMachine.stateTransition.abort THEN
				gSuperTrak.skill.Outfeed.state.stateMachine.operationalState := ABORTING;

			ELSIF gSuperTrak.skill.Outfeed.state.stateMachine.stateTransition.stop THEN
				gSuperTrak.skill.Outfeed.state.stateMachine.operationalState := STOPPING;

			ELSE
				Outfeed_Starting;

			END_IF;

		(*************************************************************************************************)
		(* RUNNING *)
		RUNNING:

			gSuperTrak.skill.Outfeed.state.stateMachine.stateTransition.start := FALSE;

			IF gSuperTrak.skill.Outfeed.state.stateMachine.stateTransition.abort THEN
				gSuperTrak.skill.Outfeed.state.stateMachine.operationalState := ABORTING;

			ELSIF gSuperTrak.skill.Outfeed.state.stateMachine.stateTransition.stop THEN
				gSuperTrak.skill.Outfeed.state.stateMachine.operationalState := STOPPING;

			ELSIF gSuperTrak.skill.Outfeed.state.stateMachine.stateTransition.hold THEN

				gSuperTrak.skill.Outfeed.state.stateMachine.operationalState := HOLDING;

			ELSIF gSuperTrak.skill.Outfeed.state.stateMachine.stateTransition.suspend THEN

				//				gSuperTrak.skill.Outfeed.state.stateMachine.operationalState := SUSPENDING;

			ELSIF gSuperTrak.skill.Outfeed.state.stateMachine.stateTransition.pause THEN

				//				gSuperTrak.skill.Outfeed.state.stateMachine.operationalState := PAUSING;

			ELSE
				Outfeed_Running;

			END_IF;

		(*************************************************************************************************)
		(* PAUSING *)
		PAUSING:
			(*gSuperTrak.skill.Outfeed.state.stateMachine.stateTransition.pause := FALSE;*)

			IF gSuperTrak.skill.Outfeed.state.stateMachine.stateTransition.abort THEN
				gSuperTrak.skill.Outfeed.state.stateMachine.operationalState := ABORTING;

			ELSIF gSuperTrak.skill.Outfeed.state.stateMachine.stateTransition.stop THEN
				gSuperTrak.skill.Outfeed.state.stateMachine.operationalState := STOPPING;

			ELSIF gSuperTrak.skill.Outfeed.state.stateMachine.stateTransition.hold THEN

				//				gSuperTrak.skill.Outfeed.state.stateMachine.operationalState := HOLDING;

			ELSIF gSuperTrak.skill.Outfeed.state.stateMachine.stateTransition.suspend THEN

				//				gSuperTrak.skill.Outfeed.state.stateMachine.operationalState := SUSPENDING;

			ELSE
				Outfeed_Pausing;
			END_IF;

		(*************************************************************************************************)
		(* PAUSED *)
		PAUSED:

			gSuperTrak.skill.Outfeed.state.stateMachine.stateTransition.pause := FALSE;

			IF gSuperTrak.skill.Outfeed.state.stateMachine.stateTransition.abort THEN
				gSuperTrak.skill.Outfeed.state.stateMachine.operationalState := ABORTING;

			ELSIF gSuperTrak.skill.Outfeed.state.stateMachine.stateTransition.stop THEN
				gSuperTrak.skill.Outfeed.state.stateMachine.operationalState := STOPPING;

			ELSIF gSuperTrak.skill.Outfeed.state.stateMachine.stateTransition.hold THEN

				//				gSuperTrak.skill.Outfeed.state.stateMachine.operationalState := HOLDING;

			ELSIF gSuperTrak.skill.Outfeed.state.stateMachine.stateTransition.suspend THEN

				//				gSuperTrak.skill.Outfeed.state.stateMachine.operationalState := SUSPENDING;

			ELSE
				Outfeed_Paused;

			END_IF;

		(*************************************************************************************************)
		(* SUSPENDING *)
		SUSPENDING:
			(*gSuperTrak.skill.Outfeed.state.stateMachine.stateTransition.suspend := FALSE;*)

			IF gSuperTrak.skill.Outfeed.state.stateMachine.stateTransition.abort THEN
				gSuperTrak.skill.Outfeed.state.stateMachine.operationalState := ABORTING;

			ELSIF gSuperTrak.skill.Outfeed.state.stateMachine.stateTransition.stop THEN
				gSuperTrak.skill.Outfeed.state.stateMachine.operationalState := STOPPING;

			ELSIF gSuperTrak.skill.Outfeed.state.stateMachine.stateTransition.hold THEN

				//				gSuperTrak.skill.Outfeed.state.stateMachine.operationalState := HOLDING;

			ELSE
				Outfeed_Suspending;

			END_IF;

		(*************************************************************************************************)
		(* SUSPENDED *)
		SUSPENDED:

			gSuperTrak.skill.Outfeed.state.stateMachine.stateTransition.suspend := FALSE;

			IF gSuperTrak.skill.Outfeed.state.stateMachine.stateTransition.abort THEN
				gSuperTrak.skill.Outfeed.state.stateMachine.operationalState := ABORTING;

			ELSIF gSuperTrak.skill.Outfeed.state.stateMachine.stateTransition.stop THEN
				gSuperTrak.skill.Outfeed.state.stateMachine.operationalState := STOPPING;

			ELSIF gSuperTrak.skill.Outfeed.state.stateMachine.stateTransition.hold THEN

				//				gSuperTrak.skill.Outfeed.state.stateMachine.operationalState := HOLDING;

			ELSE
				Outfeed_Suspended;

			END_IF;

		(*************************************************************************************************)
		(* UNSUSPENDING *)
		UNSUSPENDING:
			gSuperTrak.skill.Outfeed.state.stateMachine.stateTransition.unsuspend := FALSE;

			IF gSuperTrak.skill.Outfeed.state.stateMachine.stateTransition.abort THEN
				gSuperTrak.skill.Outfeed.state.stateMachine.operationalState := ABORTING;

			ELSIF gSuperTrak.skill.Outfeed.state.stateMachine.stateTransition.stop THEN
				gSuperTrak.skill.Outfeed.state.stateMachine.operationalState := STOPPING;

			ELSIF gSuperTrak.skill.Outfeed.state.stateMachine.stateTransition.hold THEN

				//				gSuperTrak.skill.Outfeed.state.stateMachine.operationalState := HOLDING;

			ELSE
				Outfeed_Unsuspending;

			END_IF;

		(*************************************************************************************************)
		(* HOLDING *)
		HOLDING:
			(*gSuperTrak.skill.Outfeed.state.stateMachine.stateTransition.hold := FALSE;*)

			IF gSuperTrak.skill.Outfeed.state.stateMachine.stateTransition.abort THEN
				gSuperTrak.skill.Outfeed.state.stateMachine.operationalState := ABORTING;

			ELSIF gSuperTrak.skill.Outfeed.state.stateMachine.stateTransition.stop THEN
				gSuperTrak.skill.Outfeed.state.stateMachine.operationalState := STOPPING;

			ELSE
				Outfeed_Holding;

			END_IF;

		(*************************************************************************************************)
		(* HELD *)
		HELD:

			gSuperTrak.skill.Outfeed.state.stateMachine.stateTransition.hold := FALSE;

			IF gSuperTrak.skill.Outfeed.state.stateMachine.stateTransition.abort THEN
				gSuperTrak.skill.Outfeed.state.stateMachine.operationalState := ABORTING;

			ELSIF gSuperTrak.skill.Outfeed.state.stateMachine.stateTransition.stop THEN
				gSuperTrak.skill.Outfeed.state.stateMachine.operationalState := STOPPING;

			ELSE
				Outfeed_Held;

			END_IF;

		(*************************************************************************************************)
		(* UNHOLDING *)
		UNHOLDING:
			gSuperTrak.skill.Outfeed.state.stateMachine.stateTransition.unhold := FALSE;

			IF gSuperTrak.skill.Outfeed.state.stateMachine.stateTransition.abort THEN
				gSuperTrak.skill.Outfeed.state.stateMachine.operationalState := ABORTING;

			ELSIF gSuperTrak.skill.Outfeed.state.stateMachine.stateTransition.stop THEN
				gSuperTrak.skill.Outfeed.state.stateMachine.operationalState := STOPPING;

			ELSE
				Outfeed_Unholding;

			END_IF;

		(*************************************************************************************************)
		(* COMPLETING *)
		COMPLETING:

			IF gSuperTrak.skill.Outfeed.state.stateMachine.stateTransition.abort THEN
				gSuperTrak.skill.Outfeed.state.stateMachine.operationalState := ABORTING;

			ELSIF gSuperTrak.skill.Outfeed.state.stateMachine.stateTransition.stop THEN
				gSuperTrak.skill.Outfeed.state.stateMachine.operationalState := STOPPING;

			ELSE
				Outfeed_Completing;

			END_IF;

		(*************************************************************************************************)
		(* COMPLETE *)
		COMPLETE:

			IF gSuperTrak.skill.Outfeed.state.stateMachine.stateTransition.abort THEN
				gSuperTrak.skill.Outfeed.state.stateMachine.operationalState := ABORTING;

			ELSIF gSuperTrak.skill.Outfeed.state.stateMachine.stateTransition.stop THEN
				gSuperTrak.skill.Outfeed.state.stateMachine.operationalState := STOPPING;

			ELSE
				Outfeed_Complete;

			END_IF;

		(*************************************************************************************************)
		(* STOPPING *)
		STOPPING:
//			gSuperTrak.skill.Outfeed.state.stateMachine.stateTransition.stop := FALSE;

			IF gSuperTrak.skill.Outfeed.state.stateMachine.stateTransition.abort THEN
				gSuperTrak.skill.Outfeed.state.stateMachine.operationalState := ABORTING;

			ELSE
				Outfeed_Stopping;

			END_IF;

		(*************************************************************************************************)
		(* STOPPED *)
		STOPPED:

			gSuperTrak.skill.Outfeed.state.stateMachine.stateTransition.stop := FALSE;

			IF gSuperTrak.skill.Outfeed.state.stateMachine.stateTransition.abort THEN
				gSuperTrak.skill.Outfeed.state.stateMachine.operationalState := ABORTING;

			ELSE
				Outfeed_Stopped;

			END_IF;

		(*************************************************************************************************)
		(* ABORTING *)
		ABORTING:
			(*gSuperTrak.skill.Outfeed.state.stateMachine.stateTransition.abort := FALSE;*)

			Outfeed_Aborting;

		(*************************************************************************************************)
		(* ABORTED *)
		ABORTED:

			gSuperTrak.skill.Outfeed.state.stateMachine.stateTransition.abort := FALSE;

			Outfeed_Aborted;

		(*************************************************************************************************)
		(* CLEARING *)
		CLEARING:
			gSuperTrak.skill.Outfeed.state.stateMachine.stateTransition.clear := FALSE;

			Outfeed_Clearing;

			(*************************************************************************************************)
			(* ELSE *)
		ELSE;

	END_CASE;
END_ACTION
```

#### Outfeed_Aborting.st
```iecst
ACTION Outfeed_Aborting:

//	IF NOT Transition_From_Stopped AND gSuperTrak.state.stateMachine.operationalState <> ABORTING THEN
//		Event_Code := 77;
//		EventLog.Commands.WriteUserEvent := TRUE;
//	END_IF;
//

	//Not knowing if any trigger was set to true before the abort we make sure every one of them is false before going to aborted
	gSuperTrak.skill.Outfeed.state.stateMachine.stateTransition.abort 		:= FALSE;
	gSuperTrak.skill.Outfeed.state.stateMachine.stateTransition.clear 		:= FALSE;
	gSuperTrak.skill.Outfeed.state.stateMachine.stateTransition.hold 		:= FALSE;
	gSuperTrak.skill.Outfeed.state.stateMachine.stateTransition.pause 		:= FALSE;
	gSuperTrak.skill.Outfeed.state.stateMachine.stateTransition.reset 		:= FALSE;
	gSuperTrak.skill.Outfeed.state.stateMachine.stateTransition.resume 		:= FALSE;
	gSuperTrak.skill.Outfeed.state.stateMachine.stateTransition.start 		:= FALSE;
	gSuperTrak.skill.Outfeed.state.stateMachine.stateTransition.stop 		:= FALSE;
	gSuperTrak.skill.Outfeed.state.stateMachine.stateTransition.suspend 	:= FALSE;
	gSuperTrak.skill.Outfeed.state.stateMachine.stateTransition.unhold 		:= FALSE;
	gSuperTrak.skill.Outfeed.state.stateMachine.stateTransition.unsuspend 	:= FALSE;

	//TODO: Insert Outfeed LED Light control
	Outfeed_LED_Blue := FALSE;
	Outfeed_LED_Green := FALSE;
	Outfeed_LED_Red := TRUE;

	Outfeed_Actuator_UP := FALSE;
	Outfeed_Actuator_DOWN := FALSE;
	Outfeed_Actuator_FRONT := FALSE;
	Outfeed_Actuator_BACK := FALSE;

	Skills_Aborted := Skills_Aborted + 1;
	gSuperTrak.skill.Outfeed.state.stateMachine.operationalState := ABORTED;

END_ACTION
```
